KUKA KRL program: MyProgram_176().src

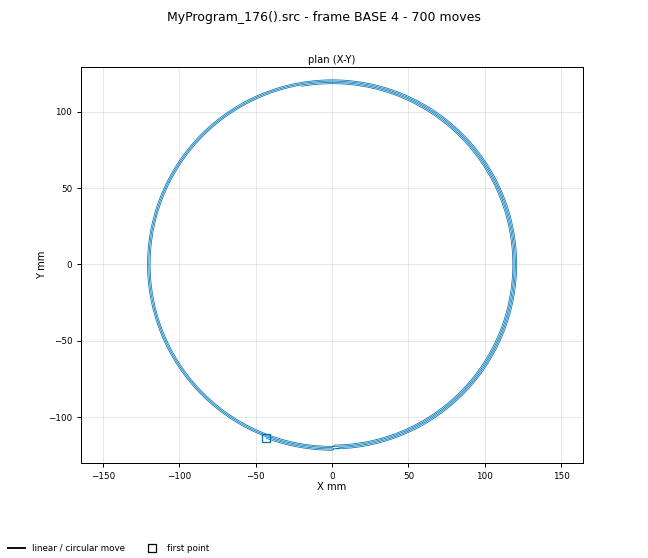
[picture p0: tool path of MyProgram_176().src in frame BASE 4, 700 of 700 moves have a stored position in this frame; points joined in program order, loops and branches not executed]
&ACCESS RVP
&REL 1
&PARAM TEMPLATE = C:\KRC\Roboter\Template\vorgabe
&PARAM EDITMASK = *
DEF MyProgram_176()
; ---- Setting reference (Base) ----
$BASE = BASE_DATA[4]

; --------------------------
; ---- Setting tool (TCP) ----
$TOOL = TOOL_DATA[3]
; --------------------------

$VEL.CP = VEL_APROX_PRINT
Startdeposition()
$VEL.CP = VEL_PRINT
LIN {X -43.076,Y -113.8011,Z 130,A -113.7942,B 24.96,C -1.4605,E1 24.9447,E2 199.9946} C_DIS
LIN {X -39.4863,Y -115.0977,Z 130,A -111.877,B 24.9598,C -1.4645,E1 24.9497,E2 198.0642} C_DIS
LIN {X -36.179,Y -116.1781,Z 130,A -110.3938,B 24.9603,C -1.456,E1 24.9536,E2 196.5985} C_DIS
LIN {X -33.1544,Y -117.077,Z 130,A -108.8854,B 24.9603,C -1.456,E1 24.9577,E2 195.0875} C_DIS
LIN {X -29.6431,Y -118.0168,Z 130,A -107.2113,B 24.9604,C -1.4532,E1 24.9622,E2 193.4176} C_DIS
LIN {X -24.0102,Y -119.2894,Z 130,A -104.7237,B 24.9611,C -1.4411,E1 24.969,E2 190.9557} C_DIS
LIN {X -19.571,Y -120.0977,Z 130,A -102.1105,B 24.9599,C -1.4632,E1 24.9763,E2 188.2874} C_DIS
LIN {X -15.3985,Y -120.7029,Z 130,A -100.2883,B 24.9603,C -1.4551,E1 24.9812,E2 186.483} C_DIS
LIN {X -11.6327,Y -121.1244,Z 130,A -98.1925,B 24.9595,C -1.4697,E1 24.9872,E2 184.3515} C_DIS
LIN {X -8.4115,Y -121.39,Z 130,A -96.7197,B 24.9597,C -1.4674,E1 24.9913,E2 182.8836} C_DIS
LIN {X -3.5905,Y -121.628,Z 130,A -94.6977,B 24.9603,C -1.4557,E1 24.9968,E2 180.8889} C_DIS
LIN {X 0.5177,Y -121.68,Z 130,A -92.4255,B 24.9594,C -1.4722,E1 25.0033,E2 178.5776} C_DIS
LIN {X 0.5177,Y -121.68,Z 130,A -92.4255,B 24.9594,C -1.4722,E1 25.0033,E2 178.5776} C_DIS
Enddeposition()
LIN {X 0.8369,Y -120.8207,Z 130,A -92.2498,B 24.9585,C -1.4882,E1 25.0039,E2 178.364} C_DIS
Startdeposition()
$VEL.CP = VEL_PRINT
LIN {X -2.018,Y -120.82,Z 130,A -95.2101,B 24.9626,C -1.4125,E1 24.9951,E2 181.5038} C_DIS
LIN {X -5.9668,Y -120.6914,Z 130,A -96.5642,B 24.9614,C -1.4362,E1 24.9915,E2 182.8019} C_DIS
LIN {X -11.9573,Y -120.2453,Z 130,A -99.4251,B 24.9614,C -1.4357,E1 24.9835,E2 185.6653} C_DIS
LIN {X -16.915,Y -119.647,Z 130,A -101.5899,B 24.9609,C -1.4455,E1 24.9776,E2 187.8085} C_DIS
LIN {X -21.3625,Y -118.9334,Z 130,A -103.8904,B 24.9612,C -1.4385,E1 24.9712,E2 190.1275} C_DIS
LIN {X -24.4172,Y -118.3441,Z 130,A -105.8718,B 24.9624,C -1.416,E1 24.9656,E2 192.1646} C_DIS
LIN {X -28.0566,Y -117.536,Z 130,A -107.1213,B 24.9611,C -1.4405,E1 24.9624,E2 193.3577} C_DIS
LIN {X -31.1677,Y -116.7485,Z 130,A -108.8063,B 24.9615,C -1.434,E1 24.9578,E2 195.0606} C_DIS
LIN {X -34.3363,Y -115.8557,Z 130,A -110.3107,B 24.9613,C -1.4376,E1 24.9537,E2 196.5589} C_DIS
LIN {X -37.706,Y -114.8044,Z 130,A -111.9297,B 24.9611,C -1.4414,E1 24.9495,E2 198.1718} C_DIS
LIN {X -40.6783,Y -113.7862,Z 130,A -113.4732,B 24.9611,C -1.4402,E1 24.9454,E2 199.721} C_DIS
LIN {X -43.9375,Y -112.5659,Z 130,A -115.4402,B 24.9618,C -1.4276,E1 24.9402,E2 201.7223} C_DIS
LIN {X -49.7061,Y -110.14,Z 130,A -117.7533,B 24.9601,C -1.4602,E1 24.9344,E2 203.9632} C_DIS
LIN {X -52.0013,Y -109.0758,Z 130,A -119.3884,B 24.961,C -1.442,E1 24.9302,E2 205.6457} C_DIS
LIN {X -54.9311,Y -107.6294,Z 130,A -120.8907,B 24.9608,C -1.4461,E1 24.9264,E2 207.1424} C_DIS
LIN {X -58.4415,Y -105.7658,Z 130,A -122.8898,B 24.961,C -1.4435,E1 24.9215,E2 209.1532} C_DIS
LIN {X -61.5431,Y -103.9902,Z 130,A -124.4503,B 24.9605,C -1.452,E1 24.9178,E2 210.6983} C_DIS
LIN {X -64.6206,Y -102.1086,Z 130,A -126.2169,B 24.9605,C -1.452,E1 24.9135,E2 212.4702} C_DIS
LIN {X -67.6234,Y -100.1429,Z 130,A -128.12,B 24.9608,C -1.4459,E1 24.9091,E2 214.3942} C_DIS
LIN {X -73.1245,Y -96.2018,Z 130,A -131.049,B 24.9599,C -1.4639,E1 24.9026,E2 217.2909} C_DIS
LIN {X -75.551,Y -94.3082,Z 130,A -132.6389,B 24.96,C -1.4608,E1 24.899,E2 218.894} C_DIS
LIN {X -78.3065,Y -92.0305,Z 130,A -134.2664,B 24.9597,C -1.4671,E1 24.8956,E2 220.5127} C_DIS
LIN {X -81.1215,Y -89.5618,Z 130,A -136.1792,B 24.9598,C -1.4646,E1 24.8916,E2 222.4392} C_DIS
LIN {X -86.9936,Y -83.8667,Z 130,A -140.8175,B 24.9612,C -1.4401,E1 24.8823,E2 227.1554} C_DIS
LIN {X -90.88,Y -79.639,Z 130,A -142.4074,B 24.9581,C -1.4954,E1 24.8795,E2 228.6207} C_DIS
LIN {X -93.2319,Y -76.8735,Z 130,A -144.4338,B 24.9586,C -1.4861,E1 24.8758,E2 230.6786} C_DIS
LIN {X -97.1767,Y -71.8227,Z 130,A -147.3387,B 24.9579,C -1.4993,E1 24.8709,E2 233.5657} C_DIS
LIN {X -99.5352,Y -68.5169,Z 130,A -149.6462,B 24.9585,C -1.4877,E1 24.8671,E2 235.9122} C_DIS
LIN {X -101.9814,Y -64.8198,Z 130,A -151.6132,B 24.9579,C -1.499,E1 24.8642,E2 237.8621} C_DIS
LIN {X -104.4534,Y -60.7555,Z 130,A -153.9133,B 24.9577,C -1.5032,E1 24.8609,E2 240.1642} C_DIS
LIN {X -106.4444,Y -57.1955,Z 130,A -155.7453,B 24.9571,C -1.5129,E1 24.8584,E2 241.9827} C_DIS
LIN {X -108.1879,Y -53.823,Z 130,A -157.6003,B 24.957,C -1.5157,E1 24.8561,E2 243.8411} C_DIS
LIN {X -109.6658,Y -50.7445,Z 130,A -159.2513,B 24.9568,C -1.5189,E1 24.8541,E2 245.4933} C_DIS
LIN {X -111.2874,Y -47.0815,Z 130,A -161.1444,B 24.9564,C -1.5247,E1 24.852,E2 247.383} C_DIS
LIN {X -112.7082,Y -43.5751,Z 130,A -163.6346,B 24.9578,C -1.5005,E1 24.8494,E2 249.945} C_DIS
LIN {X -114.4356,Y -38.808,Z 130,A -165.0376,B 24.955,C -1.5503,E1 24.8483,E2 251.2373} C_DIS
LIN {X -115.1671,Y -36.5852,Z 130,A -167.6071,B 24.9583,C -1.4919,E1 24.846,E2 253.9606} C_DIS
LIN {X -117.1214,Y -29.7357,Z 130,A -169.9378,B 24.9552,C -1.5464,E1 24.8444,E2 256.1751} C_DIS
LIN {X -118.0083,Y -25.9928,Z 130,A -171.6634,B 24.9546,C -1.5563,E1 24.8433,E2 257.8873} C_DIS
LIN {X -118.6987,Y -22.6313,Z 130,A -173.3036,B 24.9544,C -1.5609,E1 24.8424,E2 259.5262} C_DIS
LIN {X -119.3798,Y -18.7095,Z 130,A -175.2073,B 24.954,C -1.5662,E1 24.8416,E2 261.4286} C_DIS
LIN {X -119.8325,Y -15.5464,Z 130,A -176.7508,B 24.9538,C -1.5698,E1 24.841,E2 262.9726} C_DIS
LIN {X -120.266,Y -11.7482,Z 130,A -178.6463,B 24.9537,C -1.5722,E1 24.8404,E2 264.8739} C_DIS
LIN {X -120.579,Y -7.8922,Z 130,A 179.5994,B 24.9531,C -1.5815,E1 24.8401,E2 266.6164} C_DIS
LIN {X -120.773,Y -3.9289,Z 130,A 177.6956,B 24.9528,C -1.5867,E1 24.8398,E2 268.5194} C_DIS
LIN {X -120.8353,Y -0.6199,Z 130,A 176.1132,B 24.9526,C -1.5913,E1 24.8398,E2 270.1004} C_DIS
LIN {X -120.8018,Y 2.9915,Z 130,A 174.3412,B 24.9524,C -1.5943,E1 24.8398,E2 271.8758} C_DIS
LIN {X -120.6507,Y 6.7033,Z 130,A 172.6318,B 24.9519,C -1.6023,E1 24.8401,E2 273.5764} C_DIS
LIN {X -120.4096,Y 10.165,Z 130,A 171.0115,B 24.9515,C -1.6087,E1 24.8404,E2 275.1911} C_DIS
LIN {X -120.0476,Y 13.7896,Z 130,A 169.1905,B 24.9515,C -1.6104,E1 24.841,E2 277.019} C_DIS
LIN {X -119.5697,Y 17.459,Z 130,A 167.5122,B 24.9509,C -1.6194,E1 24.8416,E2 278.686} C_DIS
LIN {X -119.0095,Y 20.9396,Z 130,A 165.7537,B 24.9508,C -1.6212,E1 24.8424,E2 280.4507} C_DIS
LIN {X -118.3157,Y 24.5557,Z 130,A 164.0299,B 24.9504,C -1.6278,E1 24.8434,E2 282.169} C_DIS
LIN {X -117.5984,Y 27.7942,Z 130,A 161.4095,B 24.9527,C -1.589,E1 24.8452,E2 284.8972} C_DIS
LIN {X -115.9552,Y 34.0007,Z 130,A 159.4245,B 24.9494,C -1.643,E1 24.8466,E2 286.7648} C_DIS
LIN {X -114.9836,Y 37.1522,Z 130,A 157.0631,B 24.9512,C -1.6145,E1 24.8487,E2 289.2078} C_DIS
LIN {X -113.2851,Y 42.0534,Z 130,A 155.3822,B 24.9487,C -1.6549,E1 24.8502,E2 290.8019} C_DIS
LIN {X -111.7939,Y 45.8667,Z 130,A 153.299,B 24.9487,C -1.6549,E1 24.8523,E2 292.8966} C_DIS
LIN {X -108.0583,Y 54.0846,Z 130,A 149.0993,B 24.9477,C -1.6714,E1 24.8573,E2 297.0801} C_DIS
LIN {X -104.2609,Y 61.0851,Z 130,A 145.3907,B 24.9468,C -1.6854,E1 24.8622,E2 300.7749} C_DIS
LIN {X -102.0913,Y 64.6486,Z 130,A 143.1221,B 24.9472,C -1.6787,E1 24.8656,E2 303.0709} C_DIS
LIN {X -98.4997,Y 69.9955,Z 130,A 140.4576,B 24.9456,C -1.7039,E1 24.8697,E2 305.6885} C_DIS
LIN {X -95.4665,Y 74.0798,Z 130,A 137.7866,B 24.9459,C -1.6994,E1 24.8742,E2 308.3832} C_DIS
LIN {X -92.1592,Y 78.1555,Z 130,A 135.5093,B 24.9449,C -1.7151,E1 24.8782,E2 310.6337} C_DIS
LIN {X -88.759,Y 81.9971,Z 130,A 132.9,B 24.9449,C -1.7137,E1 24.883,E2 313.2579} C_DIS
LIN {X -86.6773,Y 84.1949,Z 130,A 131.0333,B 24.9459,C -1.6988,E1 24.8867,E2 315.1682} C_DIS
LIN {X -84.3268,Y 86.55,Z 130,A 129.5286,B 24.9455,C -1.7058,E1 24.8897,E2 316.6627} C_DIS
LIN {X -80.1655,Y 90.4176,Z 130,A 127.1282,B 24.9443,C -1.7247,E1 24.8946,E2 319.0276} C_DIS
LIN {X -77.6232,Y 92.6089,Z 130,A 124.9087,B 24.9458,C -1.7013,E1 24.8995,E2 321.3113} C_DIS
LIN {X -74.2223,Y 95.3568,Z 130,A 123.3101,B 24.9442,C -1.7262,E1 24.9029,E2 322.8566} C_DIS
LIN {X -71.5131,Y 97.4034,Z 130,A 121.4611,B 24.9446,C -1.7193,E1 24.9071,E2 324.7286} C_DIS
LIN {X -67.8075,Y 100.0183,Z 130,A 119.6468,B 24.9434,C -1.7382,E1 24.9112,E2 326.5041} C_DIS
LIN {X -63.7663,Y 102.6424,Z 130,A 116.9018,B 24.9444,C -1.7226,E1 24.9177,E2 329.295} C_DIS
LIN {X -60.5945,Y 104.5468,Z 130,A 115.1497,B 24.9442,C -1.7259,E1 24.922,E2 331.0445} C_DIS
LIN {X -57.4725,Y 106.2942,Z 130,A 113.887,B 24.9428,C -1.7477,E1 24.9249,E2 332.2589} C_DIS
LIN {X -54.5356,Y 107.8315,Z 130,A 112.1726,B 24.943,C -1.7441,E1 24.9292,E2 333.9865} C_DIS
LIN {X -50.8976,Y 109.5945,Z 130,A 110.3644,B 24.9425,C -1.7519,E1 24.9337,E2 335.7808} C_DIS
LIN {X -47.2697,Y 111.2081,Z 130,A 108.4188,B 24.9425,C -1.7519,E1 24.9387,E2 337.7309} C_DIS
LIN {X -44.0241,Y 112.5319,Z 130,A 106.7996,B 24.9422,C -1.7561,E1 24.9429,E2 339.3437} C_DIS
LIN {X -37.4229,Y 114.896,Z 130,A 103.7344,B 24.9412,C -1.7718,E1 24.9509,E2 342.3776} C_DIS
LIN {X -34.8453,Y 115.7047,Z 130,A 102.1371,B 24.942,C -1.7592,E1 24.9553,E2 344.0077} C_DIS
LIN {X -31.5071,Y 116.6568,Z 130,A 100.5707,B 24.9416,C -1.7645,E1 24.9594,E2 345.5639} C_DIS
LIN {X -28.4579,Y 117.4381,Z 130,A 99.0662,B 24.9416,C -1.7654,E1 24.9635,E2 347.0683} C_DIS
LIN {X -24.8301,Y 118.2593,Z 130,A 96.1017,B 24.9449,C -1.7139,E1 24.972,E2 350.1586} C_DIS
LIN {X -17.7522,Y 119.5277,Z 130,A 93.9207,B 24.9412,C -1.7707,E1 24.9776,E2 352.2069} C_DIS
LIN {X -9.9639,Y 120.4257,Z 130,A 90.3564,B 24.9406,C -1.7796,E1 24.9875,E2 355.7521} C_DIS
LIN {X -3.9372,Y 120.7728,Z 130,A 87.429,B 24.9408,C -1.7777,E1 24.9957,E2 358.6849} C_DIS
LIN {X 2.7012,Y 120.8075,Z 130,A 84.3293,B 24.9406,C -1.7805,E1 25.0043,E2 361.778} C_DIS
LIN {X 7.9999,Y 120.5717,Z 130,A 81.8264,B 24.9406,C -1.7811,E1 25.0113,E2 364.2787} C_DIS
LIN {X 14.0154,Y 120.0212,Z 130,A 78.8352,B 24.941,C -1.7749,E1 25.0196,E2 367.2827} C_DIS
LIN {X 17.5208,Y 119.5609,Z 130,A 77.1661,B 24.941,C -1.7748,E1 25.0242,E2 368.9506} C_DIS
LIN {X 20.1208,Y 119.1499,Z 130,A 75.8476,B 24.9412,C -1.7712,E1 25.0279,E2 370.2765} C_DIS
LIN {X 25.1832,Y 118.1848,Z 130,A 73.4943,B 24.941,C -1.7742,E1 25.0343,E2 372.6198} C_DIS
LIN {X 29.3936,Y 117.2093,Z 130,A 71.2197,B 24.9418,C -1.7626,E1 25.0405,E2 374.9185} C_DIS
LIN {X 32.9591,Y 116.255,Z 130,A 69.6385,B 24.9413,C -1.7693,E1 25.0447,E2 376.4813} C_DIS
LIN {X 35.9243,Y 115.3732,Z 130,A 68.1589,B 24.9414,C -1.7676,E1 25.0487,E2 377.9623} C_DIS
LIN {X 38.9416,Y 114.3905,Z 130,A 66.502,B 24.942,C -1.7592,E1 25.0531,E2 379.6358} C_DIS
LIN {X 43.7946,Y 112.622,Z 130,A 64.3605,B 24.9412,C -1.7712,E1 25.0587,E2 381.7444} C_DIS
LIN {X 47.1534,Y 111.2571,Z 130,A 62.5315,B 24.9417,C -1.7643,E1 25.0634,E2 383.5858} C_DIS
LIN {X 49.9349,Y 110.0369,Z 130,A 61.0033,B 24.942,C -1.7585,E1 25.0673,E2 385.1239} C_DIS
LIN {X 55.6396,Y 107.2673,Z 130,A 57.8973,B 24.9426,C -1.7499,E1 25.0751,E2 388.2416} C_DIS
LIN {X 58.9636,Y 105.4742,Z 130,A 56.2743,B 24.9422,C -1.7554,E1 25.0791,E2 389.8472} C_DIS
LIN {X 63.1397,Y 103.0296,Z 130,A 54.0038,B 24.9424,C -1.7531,E1 25.0845,E2 392.1161} C_DIS
LIN {X 65.8525,Y 101.3185,Z 130,A 51.6747,B 24.945,C -1.7125,E1 25.0902,E2 394.5334} C_DIS
LIN {X 70.1284,Y 98.4049,Z 130,A 49.9947,B 24.9429,C -1.7448,E1 25.0938,E2 396.1313} C_DIS
LIN {X 72.8347,Y 96.4195,Z 130,A 48.4007,B 24.9431,C -1.7418,E1 25.0974,E2 397.7266} C_DIS
LIN {X 75.6312,Y 94.2432,Z 130,A 46.6484,B 24.9436,C -1.7352,E1 25.1012,E2 399.488} C_DIS
LIN {X 78.4927,Y 91.8719,Z 130,A 45.0197,B 24.9434,C -1.7382,E1 25.1047,E2 401.1035} C_DIS
LIN {X 83.1482,Y 87.6821,Z 130,A 42.0599,B 24.9437,C -1.7325,E1 25.1108,E2 404.0646} C_DIS
LIN {X 85.565,Y 85.3256,Z 130,A 40.3562,B 24.9443,C -1.7241,E1 25.1142,E2 405.7811} C_DIS
LIN {X 88.5194,Y 82.2578,Z 130,A 38.4664,B 24.9442,C -1.7258,E1 25.1178,E2 407.6586} C_DIS
LIN {X 90.6008,Y 79.9587,Z 130,A 36.8642,B 24.9448,C -1.7161,E1 25.1208,E2 409.2766} C_DIS
LIN {X 93.0238,Y 77.124,Z 130,A 35.1676,B 24.9448,C -1.7154,E1 25.1239,E2 410.9671} C_DIS
LIN {X 95.3788,Y 74.1936,Z 130,A 33.3668,B 24.9452,C -1.7101,E1 25.127,E2 412.7719} C_DIS
LIN {X 97.7429,Y 71.0494,Z 130,A 31.5939,B 24.9452,C -1.7099,E1 25.1299,E2 414.5367} C_DIS
LIN {X 100.4416,Y 67.1823,Z 130,A 29.3918,B 24.9455,C -1.7058,E1 25.1334,E2 416.7378} C_DIS
LIN {X 102.2908,Y 64.3292,Z 130,A 26.8559,B 24.9486,C -1.6569,E1 25.1374,E2 419.3762} C_DIS
LIN {X 105.2879,Y 59.2973,Z 130,A 25.1515,B 24.9458,C -1.7012,E1 25.1396,E2 420.9673} C_DIS
LIN {X 106.4735,Y 57.1418,Z 130,A 23.7123,B 24.9468,C -1.6846,E1 25.1415,E2 422.438} C_DIS
LIN {X 108.2142,Y 53.77,Z 130,A 21.9702,B 24.947,C -1.6824,E1 25.1437,E2 424.1762} C_DIS
LIN {X 109.7481,Y 50.5677,Z 130,A 20.4026,B 24.947,C -1.6832,E1 25.1456,E2 425.7334} C_DIS
LIN {X 111.8091,Y 45.8294,Z 130,A 18.1564,B 24.9467,C -1.686,E1 25.148,E2 427.9606} C_DIS
LIN {X 113.5739,Y 41.2615,Z 130,A 15.7506,B 24.9474,C -1.6749,E1 25.1505,E2 430.3792} C_DIS
LIN {X 114.475,Y 38.691,Z 130,A 14.3368,B 24.9481,C -1.665,E1 25.1517,E2 431.8084} C_DIS
LIN {X 115.4974,Y 35.5239,Z 130,A 12.6878,B 24.9486,C -1.6567,E1 25.1531,E2 433.4677} C_DIS
LIN {X 116.617,Y 31.6547,Z 130,A 10.8737,B 24.9486,C -1.6555,E1 25.1545,E2 435.2742} C_DIS
LIN {X 117.5248,Y 28.1025,Z 130,A 8.6393,B 24.9505,C -1.6257,E1 25.156,E2 437.5659} C_DIS
LIN {X 118.3836,Y 24.225,Z 130,A 7.661,B 24.9481,C -1.6643,E1 25.1565,E2 438.4475} C_DIS
LIN {X 118.8903,Y 21.6022,Z 130,A 5.4208,B 24.9513,C -1.6123,E1 25.1577,E2 440.7971} C_DIS
LIN {X 119.6078,Y 17.1911,Z 130,A 3.0154,B 24.9525,C -1.5916,E1 25.1587,E2 443.2372} C_DIS
LIN {X 120.3033,Y 11.3439,Z 130,A 1.391,B 24.9496,C -1.6399,E1 25.1591,E2 444.7382} C_DIS
LIN {X 120.5914,Y 7.7094,Z 130,A -0.7853,B 24.9513,C -1.6121,E1 25.1596,E2 446.9672} C_DIS
LIN {X 120.8071,Y 2.7026,Z 130,A -3.1872,B 24.9518,C -1.603,E1 25.1598,E2 449.376} C_DIS
LIN {X 120.8349,Y -0.6737,Z 130,A -5.1757,B 24.9533,C -1.5788,E1 25.1598,E2 451.4099} C_DIS
LIN {X 120.7165,Y -5.3935,Z 130,A -6.7524,B 24.9518,C -1.604,E1 25.1596,E2 452.9178} C_DIS
LIN {X 120.432,Y -9.8834,Z 130,A -9.2672,B 24.9533,C -1.5781,E1 25.1591,E2 455.4785} C_DIS
LIN {X 120.0831,Y -13.4863,Z 130,A -10.9402,B 24.9535,C -1.5746,E1 25.1585,E2 457.15} C_DIS
LIN {X 119.6677,Y -16.769,Z 130,A -12.7265,B 24.9545,C -1.5588,E1 25.1578,E2 458.9629} C_DIS
LIN {X 118.9665,Y -21.1784,Z 130,A -14.1691,B 24.9529,C -1.5852,E1 25.1572,E2 460.3351} C_DIS
LIN {X 118.405,Y -24.1205,Z 130,A -15.6612,B 24.9534,C -1.577,E1 25.1564,E2 461.8377} C_DIS
LIN {X 117.649,Y -27.5748,Z 130,A -17.2985,B 24.9536,C -1.5735,E1 25.1554,E2 463.4737} C_DIS
LIN {X 116.5549,Y -31.8843,Z 130,A -19.7071,B 24.9549,C -1.5518,E1 25.1536,E2 465.9195} C_DIS
LIN {X 115.1104,Y -36.7604,Z 130,A -21.8943,B 24.9547,C -1.5552,E1 25.1518,E2 468.0864} C_DIS
LIN {X 112.9222,Y -43.0132,Z 130,A -24.9075,B 24.9549,C -1.5516,E1 25.149,E2 471.0912} C_DIS
LIN {X 111.4747,Y -46.637,Z 130,A -27.5616,B 24.9575,C -1.5063,E1 25.1461,E2 473.8372} C_DIS
LIN {X 109.2269,Y -51.6866,Z 130,A -29.3123,B 24.9555,C -1.541,E1 25.1441,E2 475.4969} C_DIS
LIN {X 107.4928,Y -55.1985,Z 130,A -31.2357,B 24.956,C -1.5321,E1 25.1417,E2 477.431} C_DIS
LIN {X 104.5166,Y -60.647,Z 130,A -34.261,B 24.9568,C -1.5193,E1 25.1376,E2 480.4707} C_DIS
LIN {X 102.1156,Y -64.6097,Z 130,A -36.2375,B 24.9565,C -1.5238,E1 25.1347,E2 482.4266} C_DIS
LIN {X 99.789,Y -68.1462,Z 130,A -38.7448,B 24.9582,C -1.4935,E1 25.1307,E2 484.9928} C_DIS
LIN {X 97.6721,Y -71.1461,Z 130,A -40.9439,B 24.9597,C -1.4665,E1 25.127,E2 487.2452} C_DIS
LIN {X 94.0738,Y -75.8402,Z 130,A -42.8999,B 24.9578,C -1.5001,E1 25.1237,E2 489.1125} C_DIS
LIN {X 89.52,Y -81.1677,Z 130,A -46.9455,B 24.9603,C -1.4563,E1 25.1161,E2 493.2434} C_DIS
LIN {X 85.807,Y -85.0807,Z 130,A -48.6974,B 24.9585,C -1.489,E1 25.1129,E2 494.9105} C_DIS
LIN {X 81.3874,Y -89.3184,Z 130,A -51.464,B 24.9585,C -1.4887,E1 25.1073,E2 497.6666} C_DIS
LIN {X 76.2591,Y -93.7343,Z 130,A -55.6715,B 24.9615,C -1.4331,E1 25.098,E2 501.9891} C_DIS
LIN {X 71.5574,Y -97.3709,Z 130,A -57.9633,B 24.9605,C -1.4523,E1 25.093,E2 504.2273} C_DIS
LIN {X 68.6596,Y -99.436,Z 130,A -59.1332,B 24.9593,C -1.4738,E1 25.0905,E2 505.3424} C_DIS
LIN {X 66.3148,Y -101.0145,Z 130,A -60.9519,B 24.9607,C -1.448,E1 25.0861,E2 507.216} C_DIS
LIN {X 63.3988,Y -102.8704,Z 130,A -62.6823,B 24.9611,C -1.4405,E1 25.0819,E2 508.9587} C_DIS
LIN {X 60.1197,Y -104.8196,Z 130,A -63.6191,B 24.959,C -1.4792,E1 25.0799,E2 509.8012} C_DIS
LIN {X 57.4223,Y -106.3214,Z 130,A -65.3981,B 24.96,C -1.4613,E1 25.0755,E2 511.6174} C_DIS
LIN {X 54.763,Y -107.7154,Z 130,A -66.8713,B 24.9603,C -1.4565,E1 25.0718,E2 513.0978} C_DIS
LIN {X 51.9658,Y -109.0928,Z 130,A -69.5341,B 24.9634,C -1.3978,E1 25.0648,E2 515.8924} C_DIS
LIN {X 45.4408,Y -111.9672,Z 130,A -71.5249,B 24.9601,C -1.4587,E1 25.06,E2 517.7346} C_DIS
LIN {X 39.7455,Y -114.1135,Z 130,A -74.882,B 24.9616,C -1.4323,E1 25.0511,E2 521.1472} C_DIS
LIN {X 35.0777,Y -115.6357,Z 130,A -77.1138,B 24.9615,C -1.434,E1 25.0451,E2 523.3708} C_DIS
LIN {X 31.3737,Y -116.6929,Z 130,A -78.7627,B 24.9611,C -1.4404,E1 25.0407,E2 525.0018} C_DIS
LIN {X 27.4643,Y -117.6746,Z 130,A -80.6829,B 24.9613,C -1.4381,E1 25.0355,E2 526.9247} C_DIS
LIN {X 24.1785,Y -118.3931,Z 130,A -82.9029,B 24.9629,C -1.4073,E1 25.0293,E2 529.2147} C_DIS
LIN {X 19.5282,Y -119.249,Z 130,A -84.3513,B 24.961,C -1.4428,E1 25.0255,E2 530.5778} C_DIS
LIN {X 16.3727,Y -119.7233,Z 130,A -86.3388,B 24.9623,C -1.4194,E1 25.0199,E2 532.6188} C_DIS
LIN {X 13.1382,Y -120.1217,Z 130,A -87.4533,B 24.9612,C -1.4387,E1 25.0169,E2 533.6869} C_DIS
LIN {X 6.275,Y -120.6743,Z 130,A -90.7049,B 24.9612,C -1.4377,E1 25.0079,E2 536.9393} C_DIS
LIN {X 0.8369,Y -120.8207,Z 130,A -92.2444,B 24.9586,C -1.486,E1 25.004,E2 538.3639} C_DIS
Enddeposition()
LIN {X 0.8369,Y -120.8207,Z 130,A -92.2444,B 24.9586,C -1.486,E1 25.004,E2 538.3639} C_DIS
Startdeposition()
$VEL.CP = VEL_PRINT
LIN {X 6.5039,Y -119.8162,Z 130,A -88.9736,B 24.9562,C -1.5281,E1 25.0133,E2 534.9944} C_DIS
LIN {X 12.9507,Y -119.2925,Z 130,A -86.9934,B 24.9591,C -1.4771,E1 25.0184,E2 533.1363} C_DIS
LIN {X 18.4281,Y -118.5691,Z 130,A -84.139,B 24.9585,C -1.4891,E1 25.0264,E2 530.2559} C_DIS
LIN {X 23.9345,Y -117.5814,Z 130,A -81.5882,B 24.9587,C -1.4856,E1 25.0334,E2 527.7164} C_DIS
LIN {X 27.1502,Y -116.8807,Z 130,A -80.0523,B 24.9587,C -1.4854,E1 25.0375,E2 526.183} C_DIS
LIN {X 30.9453,Y -115.9342,Z 130,A -78.1094,B 24.9584,C -1.4909,E1 25.0428,E2 524.23} C_DIS
LIN {X 34.5242,Y -114.9194,Z 130,A -76.3874,B 24.9584,C -1.4904,E1 25.0474,E2 522.5124} C_DIS
LIN {X 37.3657,Y -114.0273,Z 130,A -74.1716,B 24.9561,C -1.5304,E1 25.0536,E2 520.2061} C_DIS
LIN {X 42.4968,Y -112.2151,Z 130,A -72.3887,B 24.9582,C -1.4945,E1 25.058,E2 518.5118} C_DIS
LIN {X 46.0571,Y -110.803,Z 130,A -70.5774,B 24.9581,C -1.4962,E1 25.0627,E2 516.7006} C_DIS
LIN {X 52.0417,Y -108.1198,Z 130,A -67.4338,B 24.9578,C -1.5017,E1 25.0707,E2 513.5519} C_DIS
LIN {X 55.5917,Y -106.3387,Z 130,A -65.5145,B 24.9575,C -1.506,E1 25.0754,E2 511.6276} C_DIS
LIN {X 59.4379,Y -104.2378,Z 130,A -63.6639,B 24.958,C -1.4981,E1 25.0799,E2 509.8013} C_DIS
LIN {X 61.3807,Y -103.1056,Z 130,A -61.6541,B 24.9552,C -1.5457,E1 25.085,E2 507.6851} C_DIS
LIN {X 65.7777,Y -100.3574,Z 130,A -59.8947,B 24.957,C -1.5155,E1 25.0889,E2 506.0029} C_DIS
LIN {X 69.2496,Y -97.9949,Z 130,A -57.7751,B 24.9564,C -1.5252,E1 25.0938,E2 503.8677} C_DIS
LIN {X 74.4542,Y -94.0999,Z 130,A -54.8659,B 24.9566,C -1.5224,E1 25.1003,E2 500.9757} C_DIS
LIN {X 77.3844,Y -91.7071,Z 130,A -53.1711,B 24.9566,C -1.521,E1 25.1039,E2 499.2907} C_DIS
LIN {X 79.9878,Y -89.4437,Z 130,A -51.5346,B 24.9565,C -1.5243,E1 25.1073,E2 497.6528} C_DIS
LIN {X 84.8501,Y -84.8481,Z 130,A -48.2821,B 24.9559,C -1.5348,E1 25.1139,E2 494.3889} C_DIS
LIN {X 89.5758,Y -79.8402,Z 130,A -44.353,B 24.9535,C -1.575,E1 25.1215,E2 490.3824} C_DIS
LIN {X 92.5554,Y -76.3668,Z 130,A -42.709,B 24.9548,C -1.5539,E1 25.1243,E2 488.7957} C_DIS
LIN {X 94.6457,Y -73.7621,Z 130,A -40.691,B 24.9533,C -1.5792,E1 25.1279,E2 486.7274} C_DIS
LIN {X 97.0751,Y -70.5324,Z 130,A -39.0741,B 24.9539,C -1.569,E1 25.1305,E2 485.1424} C_DIS
LIN {X 99.4513,Y -67.1393,Z 130,A -37.2891,B 24.9541,C -1.5651,E1 25.1333,E2 483.3756} C_DIS
LIN {X 101.4734,Y -64.0444,Z 130,A -35.6903,B 24.9543,C -1.5619,E1 25.1356,E2 481.7922} C_DIS
LIN {X 103.6666,Y -60.4316,Z 130,A -32.8628,B 24.9515,C -1.6081,E1 25.1398,E2 478.8703} C_DIS
LIN {X 106.0318,Y -56.1743,Z 130,A -31.2681,B 24.9533,C -1.5786,E1 25.1418,E2 477.3535} C_DIS
LIN {X 107.5334,Y -53.2428,Z 130,A -29.717,B 24.9531,C -1.5823,E1 25.1437,E2 475.8019} C_DIS
LIN {X 109.7932,Y -48.414,Z 130,A -27.2149,B 24.9528,C -1.5879,E1 25.1467,E2 473.3003} C_DIS
LIN {X 111.0584,Y -45.4345,Z 130,A -25.6302,B 24.9524,C -1.5947,E1 25.1484,E2 471.7083} C_DIS
LIN {X 112.2392,Y -42.4332,Z 130,A -24.1036,B 24.9521,C -1.5988,E1 25.1499,E2 470.1803} C_DIS
LIN {X 113.9931,Y -37.4712,Z 130,A -21.5812,B 24.9516,C -1.6072,E1 25.1522,E2 467.6524} C_DIS
LIN {X 114.9984,Y -34.2579,Z 130,A -19.9341,B 24.9512,C -1.6144,E1 25.1536,E2 465.9978} C_DIS
LIN {X 116.1617,Y -30.0784,Z 130,A -17.9335,B 24.951,C -1.6175,E1 25.155,E2 464.0013} C_DIS
LIN {X 116.9905,Y -26.6748,Z 130,A -16.1961,B 24.9505,C -1.6261,E1 25.1561,E2 462.2537} C_DIS
LIN {X 117.8009,Y -22.8292,Z 130,A -14.4442,B 24.9505,C -1.6261,E1 25.1571,E2 460.5123} C_DIS
LIN {X 118.308,Y -20.0372,Z 130,A -12.323,B 24.9478,C -1.6688,E1 25.1581,E2 458.3025} C_DIS
LIN {X 119.0724,Y -14.8432,Z 130,A -10.4886,B 24.9494,C -1.6433,E1 25.1587,E2 456.5393} C_DIS
LIN {X 119.4099,Y -11.8299,Z 130,A -8.5637,B 24.9476,C -1.6719,E1 25.1593,E2 454.5583} C_DIS
LIN {X 119.7636,Y -7.4382,Z 130,A -7.1074,B 24.9492,C -1.6464,E1 25.1596,E2 453.1708} C_DIS
LIN {X 119.9809,Y -1.7386,Z 130,A -4.3448,B 24.9485,C -1.6572,E1 25.1598,E2 450.399} C_DIS
LIN {X 119.9682,Y 2.4259,Z 130,A -1.9376,B 24.9468,C -1.6847,E1 25.1597,E2 447.9415} C_DIS
LIN {X 119.8331,Y 6.1988,Z 130,A -0.1113,B 24.9464,C -1.6917,E1 25.1594,E2 446.1094} C_DIS
LIN {X 119.565,Y 10.1366,Z 130,A 1.4041,B 24.9471,C -1.6794,E1 25.1591,E2 444.6321} C_DIS
LIN {X 119.2131,Y 13.658,Z 130,A 3.4648,B 24.9456,C -1.7034,E1 25.1584,E2 442.527} C_DIS
LIN {X 118.6785,Y 17.72,Z 130,A 5.1451,B 24.9461,C -1.6958,E1 25.1578,E2 440.8744} C_DIS
LIN {X 117.9021,Y 22.3036,Z 130,A 7.2282,B 24.9461,C -1.6961,E1 25.1567,E2 438.8029} C_DIS
LIN {X 117.3081,Y 25.2417,Z 130,A 8.7616,B 24.9455,C -1.7057,E1 25.1558,E2 437.2558} C_DIS
LIN {X 116.2726,Y 29.6471,Z 130,A 10.6727,B 24.9458,C -1.7,E1 25.1546,E2 435.369} C_DIS
LIN {X 115.4843,Y 32.5824,Z 130,A 12.165,B 24.9454,C -1.7066,E1 25.1534,E2 433.8698} C_DIS
LIN {X 114.3401,Y 36.3988,Z 130,A 14.0581,B 24.9451,C -1.7119,E1 25.1519,E2 431.9749} C_DIS
LIN {X 113.3434,Y 39.3907,Z 130,A 15.4299,B 24.9452,C -1.7099,E1 25.1507,E2 430.6157} C_DIS
LIN {X 111.559,Y 44.1918,Z 130,A 17.8886,B 24.9447,C -1.7178,E1 25.1482,E2 428.152} C_DIS
LIN {X 109.6568,Y 48.7236,Z 130,A 20.2927,B 24.9441,C -1.7275,E1 25.1456,E2 425.7383} C_DIS
LIN {X 108.1415,Y 51.9965,Z 130,A 21.9729,B 24.9439,C -1.7304,E1 25.1436,E2 424.0603} C_DIS
LIN {X 106.5374,Y 55.2129,Z 130,A 23.8202,B 24.9432,C -1.7416,E1 25.1412,E2 422.1963} C_DIS
LIN {X 104.4763,Y 59.0192,Z 130,A 26.2798,B 24.9415,C -1.7667,E1 25.1378,E2 419.6903} C_DIS
LIN {X 102.3827,Y 62.5786,Z 130,A 27.6907,B 24.943,C -1.7444,E1 25.1358,E2 418.3391} C_DIS
LIN {X 100.344,Y 65.7981,Z 130,A 29.5092,B 24.9427,C -1.7492,E1 25.1331,E2 416.5186} C_DIS
LIN {X 98.7619,Y 68.1503,Z 130,A 31.0473,B 24.9418,C -1.7617,E1 25.1306,E2 414.9586} C_DIS
LIN {X 96.0615,Y 71.9058,Z 130,A 33.0552,B 24.9421,C -1.7574,E1 25.1273,E2 412.9704} C_DIS
LIN {X 94.0524,Y 74.5143,Z 130,A 34.6417,B 24.9418,C -1.762,E1 25.1246,E2 411.3805} C_DIS
LIN {X 91.4546,Y 77.6808,Z 130,A 36.5575,B 24.9416,C -1.7647,E1 25.1212,E2 409.4672} C_DIS
LIN {X 89.3382,Y 80.1056,Z 130,A 38.1254,B 24.9413,C -1.7698,E1 25.1183,E2 407.8942} C_DIS
LIN {X 87.0907,Y 82.5447,Z 130,A 39.6353,B 24.9413,C -1.7698,E1 25.1154,E2 406.391} C_DIS
LIN {X 84.5295,Y 85.1649,Z 130,A 41.2875,B 24.9413,C -1.7689,E1 25.1122,E2 404.7479} C_DIS
LIN {X 82.0889,Y 87.5194,Z 130,A 43.5789,B 24.9389,C -1.8048,E1 25.1074,E2 402.3811} C_DIS
LIN {X 78.9295,Y 90.3789,Z 130,A 44.9931,B 24.9407,C -1.7789,E1 25.1046,E2 401.0337} C_DIS
LIN {X 76.6174,Y 92.3472,Z 130,A 46.492,B 24.9403,C -1.7841,E1 25.1013,E2 399.5284} C_DIS
LIN {X 73.5252,Y 94.8282,Z 130,A 48.4223,B 24.94,C -1.7894,E1 25.0971,E2 397.5926} C_DIS
LIN {X 70.9387,Y 96.7777,Z 130,A 49.8331,B 24.9402,C -1.7857,E1 25.094,E2 396.1957} C_DIS
LIN {X 66.9086,Y 99.6075,Z 130,A 52.3228,B 24.9395,C -1.7962,E1 25.0882,E2 393.6896} C_DIS
LIN {X 63.8499,Y 101.5948,Z 130,A 54.0245,B 24.9395,C -1.7971,E1 25.0842,E2 391.9913} C_DIS
LIN {X 61.0925,Y 103.2759,Z 130,A 55.7301,B 24.9388,C -1.8072,E1 25.0801,E2 390.2671} C_DIS
LIN {X 57.2326,Y 105.4639,Z 130,A 57.641,B 24.9392,C -1.8004,E1 25.0755,E2 388.378} C_DIS
LIN {X 54.8566,Y 106.7195,Z 130,A 59.2066,B 24.9382,C -1.8154,E1 25.0715,E2 386.781} C_DIS
LIN {X 50.687,Y 108.7614,Z 130,A 61.0821,B 24.9391,C -1.802,E1 25.0669,E2 384.9422} C_DIS
LIN {X 47.7179,Y 110.0967,Z 130,A 62.681,B 24.9389,C -1.8059,E1 25.0628,E2 383.3381} C_DIS
LIN {X 43.1826,Y 111.9554,Z 130,A 65.3462,B 24.9377,C -1.8235,E1 25.0558,E2 380.6371} C_DIS
LIN {X 38.4379,Y 113.6695,Z 130,A 67.3528,B 24.9388,C -1.8068,E1 25.0506,E2 378.6741} C_DIS
LIN {X 35.7611,Y 114.54,Z 130,A 68.7853,B 24.9385,C -1.812,E1 25.0467,E2 377.2319} C_DIS
LIN {X 32.601,Y 115.479,Z 130,A 70.4068,B 24.9382,C -1.8154,E1 25.0424,E2 375.6052} C_DIS
LIN {X 28.7137,Y 116.5067,Z 130,A 72.2699,B 24.9383,C -1.8139,E1 25.0374,E2 373.7483} C_DIS
LIN {X 25.7053,Y 117.207,Z 130,A 73.5633,B 24.9388,C -1.8063,E1 25.0339,E2 372.4748} C_DIS
LIN {X 22.1661,Y 117.9286,Z 130,A 75.4805,B 24.9382,C -1.8159,E1 25.0286,E2 370.5371} C_DIS
LIN {X 18.9583,Y 118.4871,Z 130,A 77.1564,B 24.9378,C -1.8221,E1 25.0239,E2 368.8483} C_DIS
LIN {X 15.2018,Y 119.0259,Z 130,A 78.9912,B 24.9377,C -1.8236,E1 25.0188,E2 367.0116} C_DIS
LIN {X 9.3951,Y 119.6243,Z 130,A 81.5904,B 24.9382,C -1.8152,E1 25.0117,E2 364.4337} C_DIS
LIN {X 5.4968,Y 119.8671,Z 130,A 83.5206,B 24.938,C -1.8182,E1 25.0063,E2 362.4972} C_DIS
LIN {X 1.3481,Y 119.9864,Z 130,A 85.8978,B 24.9368,C -1.836,E1 24.9995,E2 360.078} C_DIS
LIN {X -2.285,Y 119.9708,Z 130,A 87.2212,B 24.9381,C -1.8168,E1 24.996,E2 358.8002} C_DIS
LIN {X -5.8073,Y 119.8536,Z 130,A 89.3751,B 24.9367,C -1.8377,E1 24.9898,E2 356.5962} C_DIS
LIN {X -9.693,Y 119.6005,Z 130,A 90.6791,B 24.9385,C -1.8116,E1 24.9864,E2 355.3536} C_DIS
LIN {X -14.7003,Y 119.0909,Z 130,A 93.2525,B 24.9381,C -1.8179,E1 24.9792,E2 352.7636} C_DIS
LIN {X -18.644,Y 118.5357,Z 130,A 94.9707,B 24.9387,C -1.8084,E1 24.9745,E2 351.0665} C_DIS
LIN {X -24.8872,Y 117.3854,Z 130,A 98.1601,B 24.9384,C -1.8129,E1 24.9657,E2 347.8628} C_DIS
LIN {X -28.086,Y 116.6599,Z 130,A 99.6937,B 24.9386,C -1.81,E1 24.9615,E2 346.3341} C_DIS
LIN {X -31.4345,Y 115.802,Z 130,A 101.3362,B 24.9387,C -1.808,E1 24.9571,E2 344.694} C_DIS
LIN {X -35.3705,Y 114.6611,Z 130,A 103.2095,B 24.9391,C -1.8021,E1 24.9521,E2 342.8315} C_DIS
LIN {X -40.8868,Y 112.812,Z 130,A 106.0852,B 24.9391,C -1.8029,E1 24.9445,E2 339.9483} C_DIS
LIN {X -44.6679,Y 111.3704,Z 130,A 108.0753,B 24.9391,C -1.8029,E1 24.9393,E2 337.9542} C_DIS
LIN {X -47.9272,Y 110.0054,Z 130,A 109.5516,B 24.9399,C -1.791,E1 24.9356,E2 336.5025} C_DIS
LIN {X -50.6478,Y 108.7796,Z 130,A 111.0888,B 24.9397,C -1.7938,E1 24.9317,E2 334.9549} C_DIS
LIN {X -53.0354,Y 107.6361,Z 130,A 112.5162,B 24.9393,C -1.799,E1 24.928,E2 333.5115} C_DIS
LIN {X -56.9184,Y 105.6344,Z 130,A 114.5057,B 24.9399,C -1.7912,E1 24.9232,E2 331.535} C_DIS
LIN {X -64.0115,Y 101.4939,Z 130,A 118.6461,B 24.9397,C -1.7935,E1 24.9132,E2 327.3766} C_DIS
LIN {X -67.9622,Y 98.8927,Z 130,A 120.6001,B 24.9409,C -1.7756,E1 24.9087,E2 325.4585} C_DIS
LIN {X -71.4323,Y 96.4162,Z 130,A 122.6834,B 24.9411,C -1.7735,E1 24.904,E2 323.373} C_DIS
LIN {X -73.2482,Y 95.0417,Z 130,A 124.4956,B 24.9391,C -1.8029,E1 24.8999,E2 321.4842} C_DIS
LIN {X -77.0107,Y 92.0204,Z 130,A 126.2499,B 24.941,C -1.7736,E1 24.8962,E2 319.7929} C_DIS
LIN {X -79.6644,Y 89.7332,Z 130,A 127.6712,B 24.942,C -1.7589,E1 24.8933,E2 318.4011} C_DIS
LIN {X -81.6161,Y 87.9629,Z 130,A 129.1305,B 24.9416,C -1.7646,E1 24.8903,E2 316.9223} C_DIS
LIN {X -85.9107,Y 83.7738,Z 130,A 132.044,B 24.942,C -1.7597,E1 24.8845,E2 314.0082} C_DIS
LIN {X -88.1332,Y 81.4305,Z 130,A 133.443,B 24.9426,C -1.7496,E1 24.8818,E2 312.627} C_DIS
LIN {X -90.8313,Y 78.4115,Z 130,A 135.5383,B 24.9425,C -1.7516,E1 24.878,E2 310.5176} C_DIS
LIN {X -93.8714,Y 74.7433,Z 130,A 137.7851,B 24.943,C -1.7444,E1 24.874,E2 308.2776} C_DIS
LIN {X -97.3442,Y 70.1616,Z 130,A 140.5006,B 24.9435,C -1.7355,E1 24.8695,E2 305.57} C_DIS
LIN {X -100.5758,Y 65.4466,Z 130,A 143.2956,B 24.9439,C -1.7306,E1 24.8651,E2 302.7728} C_DIS
LIN {X -102.7984,Y 61.8947,Z 130,A 145.1947,B 24.9445,C -1.7205,E1 24.8624,E2 300.8881} C_DIS
LIN {X -106.1304,Y 55.987,Z 130,A 148.5188,B 24.9449,C -1.7145,E1 24.8579,E2 297.5608} C_DIS
LIN {X -107.7565,Y 52.7926,Z 130,A 151.1702,B 24.9426,C -1.7498,E1 24.8545,E2 294.811} C_DIS
LIN {X -110.2352,Y 47.4002,Z 130,A 153.2031,B 24.9454,C -1.7065,E1 24.8523,E2 292.87} C_DIS
LIN {X -111.5515,Y 44.2111,Z 130,A 154.7426,B 24.946,C -1.6968,E1 24.8507,E2 291.345} C_DIS
LIN {X -112.8535,Y 40.773,Z 130,A 157.4278,B 24.9438,C -1.7312,E1 24.8481,E2 288.5626} C_DIS
LIN {X -114.6975,Y 35.2531,Z 130,A 159.2765,B 24.947,C -1.6825,E1 24.8466,E2 286.8196} C_DIS
LIN {X -116.9349,Y 26.9157,Z 130,A 163.4903,B 24.9475,C -1.673,E1 24.8436,E2 282.6038} C_DIS
LIN {X -117.7664,Y 23.0085,Z 130,A 165.4034,B 24.9479,C -1.667,E1 24.8425,E2 280.6936} C_DIS
LIN {X -118.3491,Y 19.7915,Z 130,A 167.0018,B 24.9481,C -1.6636,E1 24.8418,E2 279.0941} C_DIS
LIN {X -118.9467,Y 15.813,Z 130,A 168.9092,B 24.9486,C -1.6567,E1 24.841,E2 277.1917} C_DIS
LIN {X -119.3372,Y 12.5235,Z 130,A 170.4594,B 24.949,C -1.6502,E1 24.8406,E2 275.6477} C_DIS
LIN {X -119.6341,Y 9.2724,Z 130,A 172.1268,B 24.949,C -1.6497,E1 24.8402,E2 273.9715} C_DIS
LIN {X -119.8632,Y 5.5868,Z 130,A 173.9118,B 24.9493,C -1.6449,E1 24.8399,E2 272.1872} C_DIS
LIN {X -119.9704,Y 2.3108,Z 130,A 175.4338,B 24.9497,C -1.6379,E1 24.8398,E2 270.6726} C_DIS
LIN {X -119.9858,Y -1.4725,Z 130,A 177.3814,B 24.9497,C -1.6379,E1 24.8398,E2 268.7131} C_DIS
LIN {X -119.8796,Y -5.2064,Z 130,A 179.0507,B 24.9504,C -1.6273,E1 24.84,E2 267.0591} C_DIS
LIN {X -119.649,Y -9.0859,Z 130,A -178.9972,B 24.9504,C -1.6254,E1 24.8404,E2 265.0999} C_DIS
LIN {X -119.3025,Y -12.8558,Z 130,A -177.1768,B 24.9508,C -1.6201,E1 24.8409,E2 263.2812} C_DIS
LIN {X -118.8449,Y -16.5591,Z 130,A -175.4607,B 24.9513,C -1.6116,E1 24.8415,E2 261.5752} C_DIS
LIN {X -118.3264,Y -19.9275,Z 130,A -173.8253,B 24.9516,C -1.6068,E1 24.8422,E2 259.9416} C_DIS
LIN {X -117.6251,Y -23.7219,Z 130,A -171.9958,B 24.952,C -1.6004,E1 24.8432,E2 258.1166} C_DIS
LIN {X -116.9222,Y -26.9708,Z 130,A -170.4696,B 24.9525,C -1.5928,E1 24.8441,E2 256.5995} C_DIS
LIN {X -116.3628,Y -29.2962,Z 130,A -168.065,B 24.9494,C -1.6438,E1 24.846,E2 254.0591} C_DIS
LIN {X -114.4244,Y -36.134,Z 130,A -165.7144,B 24.9527,C -1.588,E1 24.8477,E2 251.8279} C_DIS
LIN {X -111.8828,Y -43.3675,Z 130,A -162.1254,B 24.9536,C -1.5739,E1 24.8511,E2 248.2523} C_DIS
LIN {X -110.6253,Y -46.4787,Z 130,A -160.5707,B 24.954,C -1.5672,E1 24.8528,E2 246.7051} C_DIS
LIN {X -109.2656,Y -49.5918,Z 130,A -158.8898,B 24.9541,C -1.565,E1 24.8547,E2 245.02} C_DIS
LIN {X -107.6421,Y -53.0233,Z 130,A -157.0395,B 24.9543,C -1.5615,E1 24.8569,E2 243.1682} C_DIS
LIN {X -106.0415,Y -56.1559,Z 130,A -155.5139,B 24.955,C -1.5501,E1 24.8589,E2 241.6615} C_DIS
LIN {X -104.1141,Y -59.6531,Z 130,A -153.1173,B 24.954,C -1.5661,E1 24.8622,E2 239.2141} C_DIS
LIN {X -102.451,Y -62.4664,Z 130,A -151.8703,B 24.9551,C -1.5483,E1 24.864,E2 238.0032} C_DIS
LIN {X -100.3797,Y -65.744,Z 130,A -150.2337,B 24.9559,C -1.5341,E1 24.8664,E2 236.3921} C_DIS
LIN {X -98.51,Y -68.5127,Z 130,A -148.4103,B 24.9556,C -1.5399,E1 24.8693,E2 234.5459} C_DIS
LIN {X -96.3497,Y -71.5201,Z 130,A -146.0405,B 24.9543,C -1.5619,E1 24.8733,E2 232.1123} C_DIS
LIN {X -93.5875,Y -75.0995,Z 130,A -144.4492,B 24.956,C -1.5317,E1 24.876,E2 230.5855} C_DIS
LIN {X -91.5028,Y -77.6242,Z 130,A -142.9267,B 24.9564,C -1.5262,E1 24.8787,E2 229.0691} C_DIS
LIN {X -89.693,Y -79.7093,Z 130,A -141.0655,B 24.9552,C -1.5471,E1 24.8823,E2 227.1498} C_DIS
LIN {X -86.892,Y -82.7556,Z 130,A -139.5013,B 24.9565,C -1.5244,E1 24.8852,E2 225.6326} C_DIS
LIN {X -84.9618,Y -84.7351,Z 130,A -137.6738,B 24.9553,C -1.5441,E1 24.8889,E2 223.7507} C_DIS
LIN {X -81.7702,Y -87.8192,Z 130,A -136.0282,B 24.9568,C -1.5186,E1 24.8921,E2 222.1589} C_DIS
LIN {X -79.0843,Y -90.2437,Z 130,A -134.4277,B 24.9573,C -1.5096,E1 24.8954,E2 220.5736} C_DIS
LIN {X -76.6438,Y -92.3253,Z 130,A -132.8254,B 24.9573,C -1.5097,E1 24.8989,E2 218.9647} C_DIS
LIN {X -73.4435,Y -94.8912,Z 130,A -131.1528,B 24.9582,C -1.4934,E1 24.9025,E2 217.3248} C_DIS
LIN {X -70.9822,Y -96.7458,Z 130,A -128.837,B 24.9562,C -1.5285,E1 24.9079,E2 214.9172} C_DIS
LIN {X -67.3912,Y -99.2807,Z 130,A -127.3979,B 24.9581,C -1.4954,E1 24.911,E2 213.552} C_DIS
LIN {X -65.0791,Y -100.8118,Z 130,A -125.9794,B 24.958,C -1.4975,E1 24.9144,E2 212.1239} C_DIS
LIN {X -62.7522,Y -102.2772,Z 130,A -124.6089,B 24.958,C -1.4981,E1 24.9176,E2 210.7478} C_DIS
LIN {X -59.7542,Y -104.056,Z 130,A -123.0152,B 24.9583,C -1.4925,E1 24.9215,E2 209.1626} C_DIS
LIN {X -56.5517,Y -105.8331,Z 130,A -121.1159,B 24.958,C -1.4969,E1 24.9262,E2 207.2475} C_DIS
LIN {X -53.1614,Y -107.5737,Z 130,A -119.406,B 24.9584,C -1.4896,E1 24.9304,E2 205.5503} C_DIS
LIN {X -49.554,Y -109.2826,Z 130,A -117.7521,B 24.9592,C -1.476,E1 24.9345,E2 203.9245} C_DIS
LIN {X -46.0241,Y -110.8169,Z 130,A -115.7359,B 24.9589,C -1.4821,E1 24.9397,E2 201.8893} C_DIS
LIN {X -42.8317,Y -112.0883,Z 130,A -113.9962,B 24.9587,C -1.485,E1 24.9443,E2 200.1389} C_DIS
LIN {X -39.5437,Y -113.2897,Z 130,A -112.3539,B 24.9588,C -1.4822,E1 24.9486,E2 198.5} C_DIS
LIN {X -35.885,Y -114.5016,Z 130,A -110.5251,B 24.959,C -1.4802,E1 24.9534,E2 196.6726} C_DIS
LIN {X -32.7785,Y -115.4287,Z 130,A -108.966,B 24.959,C -1.4796,E1 24.9576,E2 195.1123} C_DIS
LIN {X -29.1564,Y -116.3987,Z 130,A -107.123,B 24.959,C -1.4809,E1 24.9626,E2 193.2635} C_DIS
LIN {X -24.8022,Y -117.4033,Z 130,A -104.9025,B 24.9587,C -1.4839,E1 24.9687,E2 191.0332} C_DIS
LIN {X -21.2184,Y -118.1016,Z 130,A -103.2635,B 24.9591,C -1.4785,E1 24.9732,E2 189.4053} C_DIS
LIN {X -18.4819,Y -118.5608,Z 130,A -101.8589,B 24.9589,C -1.4818,E1 24.9771,E2 187.9916} C_DIS
LIN {X -11.9988,Y -119.3922,Z 130,A -98.8233,B 24.9591,C -1.4773,E1 24.9855,E2 184.9647} C_DIS
LIN {X -6.3429,Y -119.8251,Z 130,A -96.3451,B 24.9597,C -1.4665,E1 24.9923,E2 182.5109} C_DIS
LIN {X -0.2156,Y -119.9935,Z 130,A -93.2838,B 24.9593,C -1.4732,E1 25.0009,E2 179.4336} C_DIS
LIN {X -0.2156,Y -119.9935,Z 130,A -93.2838,B 24.9593,C -1.4732,E1 25.0009,E2 179.4336} C_DIS
Enddeposition()
LIN {X 0.8082,Y -119.1444,Z 130,A -93.2501,B 24.9597,C -1.4669,E1 25.001,E2 179.4147} C_DIS
Startdeposition()
$VEL.CP = VEL_PRINT
LIN {X -3.5599,Y -119.0952,Z 130,A -95.7995,B 24.9608,C -1.446,E1 24.9937,E2 182.0138} C_DIS
LIN {X -7.82,Y -118.8917,Z 130,A -97.5526,B 24.9601,C -1.4594,E1 24.9889,E2 183.7356} C_DIS
LIN {X -10.927,Y -118.6463,Z 130,A -99.1211,B 24.9603,C -1.4564,E1 24.9845,E2 185.3121} C_DIS
LIN {X -14.6865,Y -118.2413,Z 130,A -100.9305,B 24.9603,C -1.457,E1 24.9795,E2 187.1212} C_DIS
LIN {X -18.2664,Y -117.7399,Z 130,A -102.6876,B 24.9603,C -1.4566,E1 24.9746,E2 188.8807} C_DIS
LIN {X -22.2333,Y -117.056,Z 130,A -104.5257,B 24.96,C -1.4617,E1 24.9696,E2 190.7087} C_DIS
LIN {X -25.6925,Y -116.3457,Z 130,A -106.3962,B 24.9604,C -1.4547,E1 24.9644,E2 192.598} C_DIS
LIN {X -29.532,Y -115.4306,Z 130,A -108.2157,B 24.9601,C -1.4593,E1 24.9595,E2 194.4091} C_DIS
LIN {X -32.8257,Y -114.538,Z 130,A -109.9324,B 24.9602,C -1.457,E1 24.9549,E2 196.134} C_DIS
LIN {X -36.2563,Y -113.499,Z 130,A -111.6825,B 24.9602,C -1.457,E1 24.9502,E2 197.887} C_DIS
LIN {X -40.1688,Y -112.1753,Z 130,A -113.6169,B 24.96,C -1.461,E1 24.9451,E2 199.8156} C_DIS
LIN {X -43.265,Y -111.0161,Z 130,A -115.2013,B 24.96,C -1.4628,E1 24.941,E2 201.3992} C_DIS
LIN {X -46.6417,Y -109.6406,Z 130,A -117.0148,B 24.96,C -1.462,E1 24.9363,E2 203.2187} C_DIS
LIN {X -50.1696,Y -108.0711,Z 130,A -118.6557,B 24.9593,C -1.4737,E1 24.9322,E2 204.8359} C_DIS
LIN {X -52.3492,Y -107.0341,Z 130,A -120.043,B 24.9598,C -1.4651,E1 24.9286,E2 206.2472} C_DIS
LIN {X -56.0076,Y -105.1655,Z 130,A -122.0082,B 24.9596,C -1.4681,E1 24.9238,E2 208.2106} C_DIS
LIN {X -59.1625,Y -103.4224,Z 130,A -123.5675,B 24.9591,C -1.4782,E1 24.92,E2 209.7506} C_DIS
LIN {X -61.3895,Y -102.1176,Z 130,A -124.8327,B 24.9591,C -1.4789,E1 24.917,E2 211.0178} C_DIS
LIN {X -64.274,Y -100.3255,Z 130,A -126.5434,B 24.9591,C -1.4781,E1 24.9129,E2 212.7359} C_DIS
LIN {X -67.3841,Y -98.2661,Z 130,A -129.2413,B 24.9611,C -1.4419,E1 24.9065,E2 215.5289} C_DIS
LIN {X -72.0469,Y -94.8997,Z 130,A -131.2043,B 24.9589,C -1.4814,E1 24.9023,E2 217.4051} C_DIS
LIN {X -75.4058,Y -92.2526,Z 130,A -133.3051,B 24.9588,C -1.4833,E1 24.8977,E2 219.5092} C_DIS
LIN {X -78.1766,Y -89.9157,Z 130,A -134.9459,B 24.9583,C -1.4911,E1 24.8943,E2 221.1377} C_DIS
LIN {X -81.2797,Y -87.1217,Z 130,A -137.1466,B 24.9586,C -1.4869,E1 24.8897,E2 223.3574} C_DIS
LIN {X -84.4962,Y -84.0052,Z 130,A -139.1789,B 24.958,C -1.4967,E1 24.8857,E2 225.3748} C_DIS
LIN {X -87.1075,Y -81.2948,Z 130,A -141.138,B 24.9582,C -1.4944,E1 24.8819,E2 227.3481} C_DIS
LIN {X -89.9928,Y -78.0883,Z 130,A -143.0852,B 24.9576,C -1.5046,E1 24.8783,E2 229.2797} C_DIS
LIN {X -92.421,Y -75.1981,Z 130,A -144.5813,B 24.9566,C -1.5225,E1 24.8757,E2 230.7399} C_DIS
LIN {X -95.7789,Y -70.8739,Z 130,A -147.3909,B 24.9566,C -1.5214,E1 24.8709,E2 233.5656} C_DIS
LIN {X -97.322,Y -68.7393,Z 130,A -149.015,B 24.9573,C -1.5094,E1 24.8682,E2 235.2263} C_DIS
LIN {X -100.1094,Y -64.6107,Z 130,A -151.1944,B 24.9564,C -1.5248,E1 24.8649,E2 237.3799} C_DIS
LIN {X -102.0666,Y -61.4734,Z 130,A -153.9346,B 24.9585,C -1.4892,E1 24.8608,E2 240.219} C_DIS
LIN {X -105.0832,Y -56.1613,Z 130,A -155.9989,B 24.9559,C -1.5338,E1 24.8582,E2 242.1879} C_DIS
LIN {X -106.7706,Y -52.8808,Z 130,A -157.7964,B 24.9557,C -1.5378,E1 24.8559,E2 243.9855} C_DIS
LIN {X -108.578,Y -49.063,Z 130,A -159.7457,B 24.9552,C -1.5471,E1 24.8536,E2 245.9233} C_DIS
LIN {X -110.123,Y -45.4934,Z 130,A -161.7213,B 24.9551,C -1.5481,E1 24.8515,E2 247.9075} C_DIS
LIN {X -112.1399,Y -40.266,Z 130,A -164.4091,B 24.9546,C -1.5564,E1 24.8488,E2 250.5906} C_DIS
LIN {X -113.3609,Y -36.6832,Z 130,A -166.1998,B 24.9542,C -1.5632,E1 24.8473,E2 252.3754} C_DIS
LIN {X -114.4249,Y -33.223,Z 130,A -167.863,B 24.9537,C -1.5718,E1 24.8459,E2 254.0278} C_DIS
LIN {X -115.6031,Y -28.856,Z 130,A -170.2369,B 24.9538,C -1.5702,E1 24.8442,E2 256.4192} C_DIS
LIN {X -116.4662,Y -25.1402,Z 130,A -172.0638,B 24.9534,C -1.5763,E1 24.8431,E2 258.2423} C_DIS
LIN {X -117.233,Y -21.2793,Z 130,A -173.7387,B 24.9525,C -1.5914,E1 24.8423,E2 259.8911} C_DIS
LIN {X -117.6422,Y -18.8984,Z 130,A -175.2118,B 24.9531,C -1.5821,E1 24.8416,E2 261.3952} C_DIS
LIN {X -118.1976,Y -15.0249,Z 130,A -177.0234,B 24.9526,C -1.5911,E1 24.8409,E2 263.1962} C_DIS
LIN {X -118.6135,Y -11.2825,Z 130,A -178.7667,B 24.952,C -1.5997,E1 24.8404,E2 264.9293} C_DIS
LIN {X -118.8524,Y -8.4017,Z 130,A 179.814,B 24.9519,C -1.603,E1 24.8401,E2 266.3493} C_DIS
LIN {X -119.0469,Y -4.9205,Z 130,A 178.1259,B 24.9516,C -1.608,E1 24.8399,E2 268.0357} C_DIS
LIN {X -119.1439,Y -1.109,Z 130,A 176.3359,B 24.9511,C -1.6158,E1 24.8398,E2 269.8179} C_DIS
LIN {X -119.1373,Y 1.6995,Z 130,A 175.0927,B 24.9505,C -1.6246,E1 24.8398,E2 271.0475} C_DIS
LIN {X -119.0668,Y 4.4588,Z 130,A 173.5023,B 24.9509,C -1.618,E1 24.84,E2 272.6632} C_DIS
LIN {X -118.8752,Y 8.0638,Z 130,A 171.837,B 24.9504,C -1.6267,E1 24.8402,E2 274.318} C_DIS
LIN {X -118.5326,Y 12.1022,Z 130,A 169.8836,B 24.95,C -1.6329,E1 24.8407,E2 276.2683} C_DIS
LIN {X -118.1409,Y 15.4625,Z 130,A 168.2971,B 24.9496,C -1.6398,E1 24.8413,E2 277.8476} C_DIS
LIN {X -117.6152,Y 19.062,Z 130,A 166.4192,B 24.9496,C -1.6402,E1 24.8421,E2 279.7358} C_DIS
LIN {X -117.0129,Y 22.4572,Z 130,A 164.8568,B 24.949,C -1.6496,E1 24.8429,E2 281.2852} C_DIS
LIN {X -116.2042,Y 26.3283,Z 130,A 162.3781,B 24.9501,C -1.6319,E1 24.8444,E2 283.8206} C_DIS
LIN {X -115.209,Y 30.3929,Z 130,A 160.7724,B 24.9487,C -1.6551,E1 24.8455,E2 285.3804} C_DIS
LIN {X -114.2449,Y 33.8298,Z 130,A 159.1698,B 24.948,C -1.6653,E1 24.8467,E2 286.9678} C_DIS
LIN {X -113.3413,Y 36.7436,Z 130,A 157.3627,B 24.9486,C -1.6559,E1 24.8483,E2 288.8078} C_DIS
LIN {X -111.5694,Y 41.8184,Z 130,A 155.0633,B 24.9474,C -1.6758,E1 24.8504,E2 291.0727} C_DIS
LIN {X -110.3657,Y 44.8973,Z 130,A 153.5167,B 24.9469,C -1.6826,E1 24.852,E2 292.6118} C_DIS
LIN {X -108.1385,Y 50.0248,Z 130,A 150.7657,B 24.9466,C -1.6882,E1 24.8551,E2 295.3645} C_DIS
LIN {X -106.648,Y 53.1281,Z 130,A 149.1125,B 24.9463,C -1.6933,E1 24.8571,E2 297.0145} C_DIS
LIN {X -104.9996,Y 56.3182,Z 130,A 147.2437,B 24.9463,C -1.6925,E1 24.8596,E2 298.8951} C_DIS
LIN {X -102.3772,Y 60.954,Z 130,A 144.7055,B 24.9458,C -1.701,E1 24.8631,E2 301.4264} C_DIS
LIN {X -100.3549,Y 64.2282,Z 130,A 143.201,B 24.9445,C -1.7208,E1 24.8653,E2 302.8913} C_DIS
LIN {X -98.3686,Y 67.2327,Z 130,A 141.0919,B 24.9452,C -1.7099,E1 24.8686,E2 305.037} C_DIS
LIN {X -96.0655,Y 70.4825,Z 130,A 139.1683,B 24.9449,C -1.7149,E1 24.8718,E2 306.9581} C_DIS
LIN {X -93.588,Y 73.7405,Z 130,A 137.5696,B 24.9435,C -1.7357,E1 24.8744,E2 308.5147} C_DIS
LIN {X -89.6489,Y 78.482,Z 130,A 134.708,B 24.9427,C -1.7478,E1 24.8795,E2 311.3606} C_DIS
LIN {X -87.7369,Y 80.6138,Z 130,A 132.8929,B 24.9437,C -1.7328,E1 24.883,E2 313.2196} C_DIS
LIN {X -85.2824,Y 83.2092,Z 130,A 130.3494,B 24.9457,C -1.7025,E1 24.8881,E2 315.8461} C_DIS
LIN {X -81.4033,Y 87.0054,Z 130,A 128.447,B 24.9434,C -1.7383,E1 24.8918,E2 317.671} C_DIS
LIN {X -78.4062,Y 89.7151,Z 130,A 126.5784,B 24.9429,C -1.746,E1 24.8957,E2 319.5288} C_DIS
LIN {X -76.1966,Y 91.5993,Z 130,A 124.7951,B 24.9437,C -1.7328,E1 24.8996,E2 321.3504} C_DIS
LIN {X -73.3156,Y 93.9238,Z 130,A 123.3146,B 24.9427,C -1.7493,E1 24.9027,E2 322.7972} C_DIS
LIN {X -70.5437,Y 96.0207,Z 130,A 121.5252,B 24.9427,C -1.7478,E1 24.9068,E2 324.5964} C_DIS
LIN {X -67.2203,Y 98.3769,Z 130,A 119.7237,B 24.942,C -1.7585,E1 24.9109,E2 326.3786} C_DIS
LIN {X -64.9631,Y 99.8832,Z 130,A 118.5155,B 24.9416,C -1.7651,E1 24.9137,E2 327.575} C_DIS
LIN {X -60.5563,Y 102.6123,Z 130,A 115.3485,B 24.9432,C -1.7411,E1 24.9214,E2 330.8089} C_DIS
LIN {X -56.6571,Y 104.8157,Z 130,A 114.239,B 24.94,C -1.7896,E1 24.9238,E2 331.8063} C_DIS
LIN {X -53.7481,Y 106.338,Z 130,A 112.2237,B 24.9411,C -1.7733,E1 24.9289,E2 333.8658} C_DIS
LIN {X -50.3503,Y 107.987,Z 130,A 110.3801,B 24.9409,C -1.775,E1 24.9336,E2 335.71} C_DIS
LIN {X -46.8007,Y 109.5736,Z 130,A 108.6296,B 24.9404,C -1.783,E1 24.938,E2 337.4459} C_DIS
LIN {X -43.7871,Y 110.8111,Z 130,A 106.8289,B 24.9409,C -1.775,E1 24.9427,E2 339.2694} C_DIS
LIN {X -39.976,Y 112.2433,Z 130,A 105.0549,B 24.9402,C -1.7856,E1 24.9473,E2 341.0219} C_DIS
LIN {X -36.0833,Y 113.555,Z 130,A 102.9837,B 24.9404,C -1.7838,E1 24.9528,E2 343.1013} C_DIS
LIN {X -33.0504,Y 114.4743,Z 130,A 101.3447,B 24.9406,C -1.7805,E1 24.9573,E2 344.7508} C_DIS
LIN {X -29.5953,Y 115.4143,Z 130,A 99.8545,B 24.9398,C -1.7924,E1 24.9612,E2 346.215} C_DIS
LIN {X -25.6019,Y 116.3655,Z 130,A 97.9969,B 24.9393,C -1.7993,E1 24.9662,E2 348.0586} C_DIS
LIN {X -22.1006,Y 117.0816,Z 130,A 95.9774,B 24.9401,C -1.7875,E1 24.9718,E2 350.1083} C_DIS
LIN {X -18.8431,Y 117.6507,Z 130,A 94.3687,B 24.9401,C -1.7878,E1 24.9763,E2 351.7178} C_DIS
LIN {X -15.6721,Y 118.1138,Z 130,A 92.9053,B 24.9398,C -1.7923,E1 24.9803,E2 353.1718} C_DIS
LIN {X -11.9766,Y 118.5457,Z 130,A 91.028,B 24.94,C -1.7893,E1 24.9855,E2 355.0573} C_DIS
LIN {X -7.7553,Y 118.8961,Z 130,A 89.0924,B 24.9396,C -1.7947,E1 24.9909,E2 356.9809} C_DIS
LIN {X -3.6592,Y 119.0922,Z 130,A 87.1174,B 24.9396,C -1.7953,E1 24.9964,E2 358.955} C_DIS
LIN {X -0.03,Y 119.1502,Z 130,A 85.1157,B 24.9403,C -1.7842,E1 25.0021,E2 360.9829} C_DIS
LIN {X 4.8063,Y 119.0518,Z 130,A 83.169,B 24.9392,C -1.8014,E1 25.0074,E2 362.8884} C_DIS
LIN {X 7.8028,Y 118.8929,Z 130,A 81.818,B 24.9389,C -1.8056,E1 25.0111,E2 364.2291} C_DIS
LIN {X 9.8411,Y 118.7418,Z 130,A 80.6372,B 24.9395,C -1.7966,E1 25.0145,E2 365.4305} C_DIS
LIN {X 13.5588,Y 118.3748,Z 130,A 78.825,B 24.9395,C -1.7956,E1 25.0195,E2 367.2438} C_DIS
LIN {X 16.7941,Y 117.9589,Z 130,A 77.1604,B 24.9399,C -1.7909,E1 25.0241,E2 368.9182} C_DIS
LIN {X 20.3947,Y 117.3921,Z 130,A 75.55,B 24.9395,C -1.7967,E1 25.0285,E2 370.5132} C_DIS
LIN {X 22.88,Y 116.9315,Z 130,A 74.1989,B 24.9399,C -1.7901,E1 25.0323,E2 371.8784} C_DIS
LIN {X 26.6629,Y 116.1269,Z 130,A 72.4204,B 24.9398,C -1.7928,E1 25.0371,E2 373.648} C_DIS
LIN {X 29.7319,Y 115.3792,Z 130,A 70.9516,B 24.9397,C -1.7942,E1 25.041,E2 375.1114} C_DIS
LIN {X 33.1858,Y 114.4359,Z 130,A 69.2179,B 24.9397,C -1.7924,E1 25.0457,E2 376.8465} C_DIS
LIN {X 36.5571,Y 113.4017,Z 130,A 67.4857,B 24.94,C -1.7895,E1 25.0503,E2 378.5825} C_DIS
LIN {X 39.2241,Y 112.5072,Z 130,A 66.0579,B 24.9403,C -1.7848,E1 25.0541,E2 380.0185} C_DIS
LIN {X 43.2146,Y 111.0359,Z 130,A 63.9825,B 24.9405,C -1.7815,E1 25.0596,E2 382.0974} C_DIS
LIN {X 47.2304,Y 109.3883,Z 130,A 62.1695,B 24.9398,C -1.7918,E1 25.0642,E2 383.8816} C_DIS
LIN {X 49.6954,Y 108.2919,Z 130,A 60.8068,B 24.9401,C -1.7873,E1 25.0676,E2 385.2518} C_DIS
LIN {X 52.6887,Y 106.8658,Z 130,A 59.1029,B 24.9406,C -1.7803,E1 25.072,E2 386.9678} C_DIS
LIN {X 55.9333,Y 105.2047,Z 130,A 57.3516,B 24.9408,C -1.778,E1 25.0763,E2 388.7195} C_DIS
LIN {X 59.3925,Y 103.2903,Z 130,A 55.4732,B 24.9408,C -1.7763,E1 25.0809,E2 390.5962} C_DIS
LIN {X 62.8218,Y 101.2417,Z 130,A 53.7829,B 24.9403,C -1.7841,E1 25.0849,E2 392.2628} C_DIS
LIN {X 65.5553,Y 99.493,Z 130,A 51.9629,B 24.9413,C -1.7695,E1 25.0892,E2 394.1115} C_DIS
LIN {X 68.1705,Y 97.7198,Z 130,A 50.3988,B 24.9416,C -1.7649,E1 25.0928,E2 395.6812} C_DIS
LIN {X 71.4544,Y 95.3448,Z 130,A 48.5923,B 24.9414,C -1.7681,E1 25.0968,E2 397.4738} C_DIS
LIN {X 73.967,Y 93.409,Z 130,A 47.0281,B 24.9417,C -1.7634,E1 25.1003,E2 399.0431} C_DIS
LIN {X 77.0882,Y 90.8504,Z 130,A 45.0871,B 24.942,C -1.7596,E1 25.1045,E2 400.9856} C_DIS
LIN {X 82.9692,Y 85.5138,Z 130,A 41.3527,B 24.9422,C -1.7557,E1 25.1121,E2 404.7141} C_DIS
LIN {X 85.9562,Y 82.5102,Z 130,A 39.2286,B 24.9428,C -1.7471,E1 25.1163,E2 406.8494} C_DIS
LIN {X 88.5953,Y 79.6699,Z 130,A 37.4104,B 24.9429,C -1.7451,E1 25.1197,E2 408.6645} C_DIS
LIN {X 90.7501,Y 77.2061,Z 130,A 35.8723,B 24.9431,C -1.7431,E1 25.1225,E2 410.2003} C_DIS
LIN {X 93.047,Y 74.4251,Z 130,A 34.0159,B 24.9437,C -1.7331,E1 25.1258,E2 412.0717} C_DIS
LIN {X 95.2717,Y 71.5517,Z 130,A 32.437,B 24.9435,C -1.7368,E1 25.1285,E2 413.6343} C_DIS
LIN {X 97.4925,Y 68.4975,Z 130,A 30.4555,B 24.9443,C -1.7243,E1 25.1317,E2 415.6357} C_DIS
LIN {X 99.5438,Y 65.4782,Z 130,A 28.8196,B 24.9443,C -1.7254,E1 25.1342,E2 417.2608} C_DIS
LIN {X 101.7804,Y 61.9442,Z 130,A 26.8579,B 24.9444,C -1.7224,E1 25.1371,E2 419.2196} C_DIS
LIN {X 103.7627,Y 58.5657,Z 130,A 24.9609,B 24.9448,C -1.7166,E1 25.1398,E2 421.1206} C_DIS
LIN {X 105.362,Y 55.6346,Z 130,A 23.3794,B 24.945,C -1.7133,E1 25.1419,E2 422.7015} C_DIS
LIN {X 106.8356,Y 52.7497,Z 130,A 21.8108,B 24.9453,C -1.7084,E1 25.1438,E2 424.2734} C_DIS
LIN {X 108.5104,Y 49.213,Z 130,A 19.9469,B 24.9456,C -1.7038,E1 25.146,E2 426.138} C_DIS
LIN {X 109.9019,Y 46.0216,Z 130,A 18.3041,B 24.9458,C -1.7004,E1 25.1478,E2 427.7798} C_DIS
LIN {X 111.2261,Y 42.7248,Z 130,A 16.7143,B 24.9458,C -1.7011,E1 25.1495,E2 429.3592} C_DIS
LIN {X 112.2304,Y 40.013,Z 130,A 15.1205,B 24.9467,C -1.6871,E1 25.151,E2 430.9771} C_DIS
LIN {X 113.3966,Y 36.5728,Z 130,A 13.4598,B 24.9467,C -1.6859,E1 25.1524,E2 432.6311} C_DIS
LIN {X 114.4543,Y 33.1208,Z 130,A 11.6511,B 24.9473,C -1.6771,E1 25.1539,E2 434.4504} C_DIS
LIN {X 115.3944,Y 29.6729,Z 130,A 10.0954,B 24.9471,C -1.6796,E1 25.155,E2 435.9911} C_DIS
LIN {X 116.399,Y 25.4484,Z 130,A 8.0381,B 24.9475,C -1.6746,E1 25.1563,E2 438.0483} C_DIS
LIN {X 116.9097,Y 22.9935,Z 130,A 6.8455,B 24.9477,C -1.6714,E1 25.157,E2 439.2415} C_DIS
LIN {X 117.5138,Y 19.6687,Z 130,A 5.213,B 24.948,C -1.6659,E1 25.1578,E2 440.8776} C_DIS
LIN {X 118.0836,Y 15.905,Z 130,A 3.2692,B 24.9487,C -1.6544,E1 25.1585,E2 442.8368} C_DIS
LIN {X 118.5039,Y 12.3764,Z 130,A 1.7509,B 24.9485,C -1.6582,E1 25.159,E2 444.3372} C_DIS
LIN {X 118.7936,Y 9.1929,Z 130,A 0.1058,B 24.9491,C -1.648,E1 25.1594,E2 445.9966} C_DIS
LIN {X 119.0619,Y 4.5728,Z 130,A -2.2012,B 24.9498,C -1.6367,E1 25.1597,E2 448.3165} C_DIS
LIN {X 119.146,Y 0.7673,Z 130,A -3.8885,B 24.9498,C -1.6377,E1 25.1597,E2 449.9914} C_DIS
LIN {X 119.1132,Y -2.9638,Z 130,A -5.9073,B 24.9508,C -1.6209,E1 25.1597,E2 452.0378} C_DIS
LIN {X 118.9032,Y -7.6504,Z 130,A -8.1371,B 24.9511,C -1.6148,E1 25.1593,E2 454.2688} C_DIS
LIN {X 118.4894,Y -12.5146,Z 130,A -10.2596,B 24.9509,C -1.6181,E1 25.1588,E2 456.371} C_DIS
LIN {X 118.0455,Y -16.1844,Z 130,A -12.2242,B 24.9518,C -1.6031,E1 25.1581,E2 458.3592} C_DIS
LIN {X 117.322,Y -20.7844,Z 130,A -14.2713,B 24.9518,C -1.6052,E1 25.1571,E2 460.3895} C_DIS
LIN {X 116.6969,Y -24.0456,Z 130,A -15.8538,B 24.952,C -1.6007,E1 25.1563,E2 461.9733} C_DIS
LIN {X 115.8237,Y -27.9519,Z 130,A -17.7661,B 24.9523,C -1.595,E1 25.1551,E2 463.8878} C_DIS
LIN {X 114.9842,Y -31.2249,Z 130,A -19.309,B 24.9524,C -1.5938,E1 25.154,E2 465.4247} C_DIS
LIN {X 114.019,Y -34.5911,Z 130,A -21.1572,B 24.9532,C -1.5804,E1 25.1525,E2 467.2941} C_DIS
LIN {X 112.7479,Y -38.5291,Z 130,A -23.024,B 24.9532,C -1.5801,E1 25.1509,E2 469.1511} C_DIS
LIN {X 111.6981,Y -41.4769,Z 130,A -24.6553,B 24.9539,C -1.5691,E1 25.1493,E2 470.7989} C_DIS
LIN {X 110.491,Y -44.5894,Z 130,A -26.148,B 24.9539,C -1.5696,E1 25.1478,E2 472.2822} C_DIS
LIN {X 108.9509,Y -48.2337,Z 130,A -28.1194,B 24.9544,C -1.5604,E1 25.1456,E2 474.2647} C_DIS
LIN {X 107.1467,Y -52.1176,Z 130,A -30.1546,B 24.9547,C -1.5553,E1 25.1431,E2 476.3009} C_DIS
LIN {X 105.5086,Y -55.3563,Z 130,A -31.9803,B 24.9552,C -1.5461,E1 25.1408,E2 478.1385} C_DIS
LIN {X 103.549,Y -58.9422,Z 130,A -33.7921,B 24.9552,C -1.5477,E1 25.1383,E2 479.9372} C_DIS
LIN {X 101.5678,Y -62.2942,Z 130,A -35.6836,B 24.9555,C -1.5413,E1 25.1356,E2 481.8342} C_DIS
LIN {X 99.7833,Y -65.1149,Z 130,A -37.109,B 24.9553,C -1.5454,E1 25.1335,E2 483.2428} C_DIS
LIN {X 98.3478,Y -67.2634,Z 130,A -38.5258,B 24.9559,C -1.5334,E1 25.1312,E2 484.6808} C_DIS
LIN {X 96.4782,Y -69.9188,Z 130,A -40.1977,B 24.9565,C -1.5237,E1 25.1285,E2 486.3674} C_DIS
LIN {X 93.5542,Y -73.7832,Z 130,A -42.2943,B 24.9562,C -1.5287,E1 25.1249,E2 488.4424} C_DIS
LIN {X 91.2934,Y -76.5646,Z 130,A -44.2102,B 24.957,C -1.5148,E1 25.1215,E2 490.3823} C_DIS
LIN {X 87.2451,Y -81.1484,Z 130,A -46.9979,B 24.957,C -1.5145,E1 25.1163,E2 493.1582} C_DIS
LIN {X 84.7979,Y -83.6998,Z 130,A -48.587,B 24.957,C -1.5156,E1 25.1132,E2 494.7378} C_DIS
LIN {X 81.284,Y -87.1175,Z 130,A -51.1913,B 24.958,C -1.498,E1 25.1079,E2 497.3728} C_DIS
LIN {X 77.7203,Y -90.3119,Z 130,A -53.354,B 24.9579,C -1.4993,E1 25.1034,E2 499.524} C_DIS
LIN {X 74.7223,Y -92.8066,Z 130,A -55.2079,B 24.9581,C -1.4961,E1 25.0994,E2 501.3784} C_DIS
LIN {X 72.5056,Y -94.5481,Z 130,A -56.532,B 24.9581,C -1.4947,E1 25.0964,E2 502.7011} C_DIS
LIN {X 69.6311,Y -96.6857,Z 130,A -58.284,B 24.9584,C -1.4896,E1 25.0925,E2 504.4589} C_DIS
LIN {X 66.2919,Y -99.0056,Z 130,A -60.0804,B 24.9582,C -1.4932,E1 25.0884,E2 506.2407} C_DIS
LIN {X 61.6771,Y -101.9428,Z 130,A -62.8378,B 24.9589,C -1.4821,E1 25.0818,E2 509.0156} C_DIS
LIN {X 59.2714,Y -103.3598,Z 130,A -64.3047,B 24.9593,C -1.4737,E1 25.0782,E2 510.4978} C_DIS
LIN {X 55.4571,Y -105.4554,Z 130,A -66.1811,B 24.9589,C -1.4803,E1 25.0737,E2 512.3533} C_DIS
LIN {X 52.1176,Y -107.1467,Z 130,A -68.2076,B 24.9597,C -1.4666,E1 25.0685,E2 514.4067} C_DIS
LIN {X 47.6612,Y -109.2005,Z 130,A -70.3198,B 24.9593,C -1.4746,E1 25.0632,E2 516.4948} C_DIS
LIN {X 44.2282,Y -110.6378,Z 130,A -72.2218,B 24.9597,C -1.4667,E1 25.0582,E2 518.4112} C_DIS
LIN {X 40.3256,Y -112.1181,Z 130,A -74.3404,B 24.9601,C -1.4588,E1 25.0527,E2 520.544} C_DIS
LIN {X 35.7408,Y -113.6625,Z 130,A -76.4681,B 24.9598,C -1.4652,E1 25.0471,E2 522.6525} C_DIS
LIN {X 32.5006,Y -114.6301,Z 130,A -78.0458,B 24.9598,C -1.4656,E1 25.0428,E2 524.2265} C_DIS
LIN {X 28.785,Y -115.6204,Z 130,A -79.7679,B 24.9595,C -1.4696,E1 25.0382,E2 525.9365} C_DIS
LIN {X 25.6811,Y -116.3482,Z 130,A -81.2597,B 24.9595,C -1.47,E1 25.0342,E2 527.4252} C_DIS
LIN {X 23.6677,Y -116.7744,Z 130,A -82.3779,B 24.9599,C -1.4632,E1 25.0311,E2 528.5583} C_DIS
LIN {X 18.0342,Y -117.7758,Z 130,A -85.1669,B 24.9601,C -1.4593,E1 25.0234,E2 531.3536} C_DIS
LIN {X 14.2039,Y -118.2992,Z 130,A -86.8696,B 24.9598,C -1.4653,E1 25.0187,E2 533.0407} C_DIS
LIN {X 12.1826,Y -118.5242,Z 130,A -88.3205,B 24.961,C -1.4429,E1 25.0145,E2 534.5435} C_DIS
LIN {X 8.8812,Y -118.8185,Z 130,A -89.6953,B 24.9605,C -1.4522,E1 25.0108,E2 535.8957} C_DIS
LIN {X 3.1874,Y -119.1067,Z 130,A -92.3222,B 24.9603,C -1.4564,E1 25.0035,E2 538.5118} C_DIS
LIN {X 0.8082,Y -119.1444,Z 130,A -93.2484,B 24.9597,C -1.4662,E1 25.0009,E2 539.4148} C_DIS
Enddeposition()
LIN {X 0.8082,Y -119.1444,Z 130,A -93.2484,B 24.9597,C -1.4662,E1 25.0009,E2 539.4148} C_DIS
Startdeposition()
$VEL.CP = VEL_PRINT
LIN {X 1.4434,Y -118.2976,Z 130,A -92.5041,B 24.9578,C -1.501,E1 25.0033,E2 538.588} C_DIS
LIN {X 3.9892,Y -118.2375,Z 130,A -91.2409,B 24.9577,C -1.5028,E1 25.0068,E2 537.3208} C_DIS
LIN {X 6.8055,Y -118.1087,Z 130,A -89.8945,B 24.9577,C -1.5025,E1 25.0105,E2 535.9756} C_DIS
LIN {X 9.7874,Y -117.8992,Z 130,A -88.4612,B 24.9577,C -1.5025,E1 25.0145,E2 534.5429} C_DIS
LIN {X 13.0384,Y -117.5858,Z 130,A -86.8803,B 24.9577,C -1.5033,E1 25.0189,E2 532.9611} C_DIS
LIN {X 15.5658,Y -117.2763,Z 130,A -85.6195,B 24.9575,C -1.5055,E1 25.0224,E2 531.6963} C_DIS
LIN {X 18.4224,Y -116.8616,Z 130,A -84.254,B 24.9575,C -1.505,E1 25.0262,E2 530.3334} C_DIS
LIN {X 21.2641,Y -116.378,Z 130,A -82.8274,B 24.9575,C -1.5075,E1 25.0301,E2 528.9023} C_DIS
LIN {X 24.501,Y -115.7416,Z 130,A -81.2649,B 24.9575,C -1.5072,E1 25.0344,E2 527.3423} C_DIS
LIN {X 27.3273,Y -115.107,Z 130,A -79.8655,B 24.9574,C -1.5084,E1 25.0382,E2 525.942} C_DIS
LIN {X 29.8046,Y -114.4889,Z 130,A -78.601,B 24.9572,C -1.5111,E1 25.0416,E2 524.6732} C_DIS
LIN {X 32.492,Y -113.7551,Z 130,A -77.2723,B 24.9572,C -1.5116,E1 25.0452,E2 523.3455} C_DIS
LIN {X 35.7264,Y -112.7832,Z 130,A -75.6529,B 24.9572,C -1.5127,E1 25.0495,E2 521.7263} C_DIS
LIN {X 38.1526,Y -111.984,Z 130,A -74.4167,B 24.957,C -1.5143,E1 25.0528,E2 520.4888} C_DIS
LIN {X 41.2301,Y -110.8895,Z 130,A -72.8464,B 24.957,C -1.5158,E1 25.0569,E2 518.9181} C_DIS
LIN {X 43.9291,Y -109.8483,Z 130,A -71.4452,B 24.9568,C -1.5178,E1 25.0606,E2 517.5153} C_DIS
LIN {X 46.6017,Y -108.7414,Z 130,A -70.0484,B 24.9568,C -1.5197,E1 25.0642,E2 516.1173} C_DIS
LIN {X 48.9335,Y -107.7104,Z 130,A -68.8066,B 24.9566,C -1.522,E1 25.0673,E2 514.8733} C_DIS
LIN {X 51.8587,Y -106.3346,Z 130,A -67.2591,B 24.9566,C -1.5236,E1 25.0712,E2 513.3259} C_DIS
LIN {X 54.0563,Y -105.2325,Z 130,A -66.0192,B 24.9563,C -1.528,E1 25.0743,E2 512.079} C_DIS
LIN {X 56.7405,Y -103.8102,Z 130,A -64.5709,B 24.9562,C -1.5295,E1 25.0779,E2 510.6314} C_DIS
LIN {X 59.5734,Y -102.2127,Z 130,A -63.0372,B 24.9562,C -1.5304,E1 25.0816,E2 509.1002} C_DIS
LIN {X 62.0445,Y -100.7316,Z 130,A -61.6495,B 24.956,C -1.5327,E1 25.0849,E2 507.7114} C_DIS
LIN {X 64.1894,Y -99.3767,Z 130,A -60.4186,B 24.9558,C -1.5352,E1 25.0878,E2 506.4785} C_DIS
LIN {X 66.9253,Y -97.5573,Z 130,A -58.8389,B 24.9557,C -1.5379,E1 25.0915,E2 504.8978} C_DIS
LIN {X 70.1851,Y -95.2369,Z 130,A -56.9063,B 24.9555,C -1.5417,E1 25.0959,E2 502.963} C_DIS
LIN {X 72.219,Y -93.7033,Z 130,A -55.6826,B 24.9553,C -1.5439,E1 25.0986,E2 501.7385} C_DIS
LIN {X 74.5957,Y -91.8226,Z 130,A -54.1645,B 24.955,C -1.5496,E1 25.1019,E2 500.2127} C_DIS
LIN {X 77.0554,Y -89.7694,Z 130,A -52.657,B 24.955,C -1.551,E1 25.1051,E2 498.7077} C_DIS
LIN {X 79.8395,Y -87.3017,Z 130,A -50.8424,B 24.9546,C -1.5559,E1 25.1089,E2 496.8888} C_DIS
LIN {X 82.2302,Y -85.0537,Z 130,A -49.2378,B 24.9544,C -1.5605,E1 25.1121,E2 495.28} C_DIS
LIN {X 85.0544,Y -82.2294,Z 130,A -47.338,B 24.9542,C -1.5636,E1 25.1158,E2 493.3809} C_DIS
LIN {X 87.2691,Y -79.8751,Z 130,A -45.7707,B 24.954,C -1.5677,E1 25.1188,E2 491.8108} C_DIS
LIN {X 89.4384,Y -77.4398,Z 130,A -44.2347,B 24.9538,C -1.5697,E1 25.1217,E2 490.277} C_DIS
LIN {X 91.8012,Y -74.6222,Z 130,A -42.4394,B 24.9535,C -1.5752,E1 25.1249,E2 488.4771} C_DIS
LIN {X 93.7042,Y -72.2179,Z 130,A -40.9613,B 24.9533,C -1.5789,E1 25.1274,E2 486.9972} C_DIS
LIN {X 95.8668,Y -69.3249,Z 130,A -39.2672,B 24.9532,C -1.581,E1 25.1302,E2 485.3063} C_DIS
LIN {X 97.3615,Y -67.207,Z 130,A -38.0167,B 24.953,C -1.5844,E1 25.1322,E2 484.054} C_DIS
LIN {X 99.12,Y -64.5873,Z 130,A -36.4953,B 24.9527,C -1.5884,E1 25.1345,E2 482.5307} C_DIS
LIN {X 100.7168,Y -62.0688,Z 130,A -35.063,B 24.9525,C -1.592,E1 25.1367,E2 481.0972} C_DIS
LIN {X 102.2131,Y -59.5727,Z 130,A -33.6613,B 24.9523,C -1.5957,E1 25.1387,E2 479.6939} C_DIS
LIN {X 103.4693,Y -57.3596,Z 130,A -32.4348,B 24.9521,C -1.5991,E1 25.1403,E2 478.4657} C_DIS
LIN {X 104.837,Y -54.8198,Z 130,A -31.0807,B 24.952,C -1.6012,E1 25.1421,E2 477.1138} C_DIS
LIN {X 106.1689,Y -52.1939,Z 130,A -29.6297,B 24.9516,C -1.6068,E1 25.1439,E2 475.6575} C_DIS
LIN {X 107.4235,Y -49.5606,Z 130,A -28.1969,B 24.9513,C -1.6121,E1 25.1456,E2 474.22} C_DIS
LIN {X 108.6036,Y -46.9181,Z 130,A -26.8363,B 24.9512,C -1.6144,E1 25.1471,E2 472.8612} C_DIS
LIN {X 109.6725,Y -44.3609,Z 130,A -25.487,B 24.9509,C -1.6189,E1 25.1486,E2 471.5087} C_DIS
LIN {X 110.89,Y -41.2287,Z 130,A -23.8869,B 24.9507,C -1.6226,E1 25.1502,E2 469.9087} C_DIS
LIN {X 111.8654,Y -38.5037,Z 130,A -22.4933,B 24.9504,C -1.6267,E1 25.1515,E2 468.5135} C_DIS
LIN {X 112.6679,Y -36.0828,Z 130,A -21.2811,B 24.9502,C -1.6295,E1 25.1525,E2 467.3014} C_DIS
LIN {X 113.6243,Y -32.9535,Z 130,A -19.6925,B 24.9499,C -1.6348,E1 25.1538,E2 465.7096} C_DIS
LIN {X 114.3128,Y -30.4734,Z 130,A -18.4244,B 24.9496,C -1.6399,E1 25.1547,E2 464.4367} C_DIS
LIN {X 115.106,Y -27.3316,Z 130,A -16.8962,B 24.9494,C -1.6429,E1 25.1557,E2 462.9102} C_DIS
LIN {X 115.7409,Y -24.5044,Z 130,A -15.5024,B 24.9492,C -1.647,E1 25.1565,E2 461.5149} C_DIS
LIN {X 116.2419,Y -21.9968,Z 130,A -14.2436,B 24.9489,C -1.652,E1 25.1572,E2 460.2515} C_DIS
LIN {X 116.8023,Y -18.8051,Z 130,A -12.7136,B 24.9487,C -1.6552,E1 25.1579,E2 458.723} C_DIS
LIN {X 117.1834,Y -16.2512,Z 130,A -11.4432,B 24.9483,C -1.6603,E1 25.1584,E2 457.4481} C_DIS
LIN {X 117.5456,Y -13.3817,Z 130,A -10.0813,B 24.9482,C -1.663,E1 25.1589,E2 456.0879} C_DIS
LIN {X 117.869,Y -10.1631,Z 130,A -8.5251,B 24.9479,C -1.6676,E1 25.1593,E2 454.5301} C_DIS
LIN {X 118.1448,Y -6.1521,Z 130,A -6.592,B 24.9475,C -1.6733,E1 25.1596,E2 452.5949} C_DIS
LIN {X 118.2543,Y -3.4419,Z 130,A -5.2225,B 24.9471,C -1.6804,E1 25.1597,E2 451.217} C_DIS
LIN {X 118.3065,Y -0.0025,Z 130,A -3.634,B 24.947,C -1.682,E1 25.1597,E2 449.6341} C_DIS
LIN {X 118.2374,Y 3.9926,Z 130,A -1.6811,B 24.9465,C -1.6892,E1 25.1597,E2 447.6759} C_DIS
LIN {X 118.0856,Y 7.2221,Z 130,A -0.1602,B 24.9463,C -1.6921,E1 25.1594,E2 446.1572} C_DIS
LIN {X 117.8973,Y 9.8111,Z 130,A 1.0925,B 24.9461,C -1.696,E1 25.1591,E2 444.9028} C_DIS
LIN {X 117.5865,Y 13.0311,Z 130,A 2.6489,B 24.9458,C -1.7005,E1 25.1587,E2 443.3449} C_DIS
LIN {X 117.2768,Y 15.5617,Z 130,A 3.9048,B 24.9455,C -1.7055,E1 25.1583,E2 442.0845} C_DIS
LIN {X 116.8616,Y 18.422,Z 130,A 5.2696,B 24.9453,C -1.7083,E1 25.1577,E2 440.7211} C_DIS
LIN {X 116.3683,Y 21.3182,Z 130,A 6.7067,B 24.945,C -1.7135,E1 25.157,E2 439.2802} C_DIS
LIN {X 115.7427,Y 24.4958,Z 130,A 8.2357,B 24.9448,C -1.7166,E1 25.1561,E2 437.753} C_DIS
LIN {X 115.1085,Y 27.3209,Z 130,A 9.6245,B 24.9445,C -1.7203,E1 25.1552,E2 436.3634} C_DIS
LIN {X 114.0203,Y 31.556,Z 130,A 11.7324,B 24.9441,C -1.7264,E1 25.1537,E2 434.2532} C_DIS
LIN {X 113.3109,Y 34.01,Z 130,A 12.991,B 24.9438,C -1.7313,E1 25.1527,E2 432.9904} C_DIS
LIN {X 112.3384,Y 37.1012,Z 130,A 14.5205,B 24.9436,C -1.7341,E1 25.1514,E2 431.4629} C_DIS
LIN {X 111.5038,Y 39.5341,Z 130,A 15.794,B 24.9433,C -1.7392,E1 25.1503,E2 430.1844} C_DIS
LIN {X 110.4973,Y 42.2657,Z 130,A 17.1881,B 24.9431,C -1.7427,E1 25.1489,E2 428.7899} C_DIS
LIN {X 109.3028,Y 45.2693,Z 130,A 18.7161,B 24.9429,C -1.7455,E1 25.1473,E2 427.2639} C_DIS
LIN {X 108.2538,Y 47.7204,Z 130,A 19.9914,B 24.9427,C -1.7485,E1 25.1459,E2 425.9884} C_DIS
LIN {X 106.9498,Y 50.5782,Z 130,A 21.5114,B 24.9424,C -1.7528,E1 25.1441,E2 424.4665} C_DIS
LIN {X 105.679,Y 53.1823,Z 130,A 22.9031,B 24.9422,C -1.7562,E1 25.1423,E2 423.0741} C_DIS
LIN {X 103.8088,Y 56.7431,Z 130,A 24.871,B 24.9418,C -1.7626,E1 25.1397,E2 421.1014} C_DIS
LIN {X 102.2049,Y 59.5865,Z 130,A 26.4071,B 24.9416,C -1.7648,E1 25.1376,E2 419.5682} C_DIS
LIN {X 100.7166,Y 62.0691,Z 130,A 27.8048,B 24.9414,C -1.7683,E1 25.1356,E2 418.1692} C_DIS
LIN {X 99.353,Y 64.2263,Z 130,A 29.0099,B 24.9413,C -1.7701,E1 25.1338,E2 416.9659} C_DIS
LIN {X 97.5596,Y 66.9219,Z 130,A 30.5969,B 24.9409,C -1.7751,E1 25.1313,E2 415.3751} C_DIS
LIN {X 95.8932,Y 69.2884,Z 130,A 32.157,B 24.9402,C -1.7863,E1 25.1287,E2 413.7962} C_DIS
LIN {X 93.7034,Y 72.2189,Z 130,A 33.7527,B 24.9405,C -1.7823,E1 25.1261,E2 412.2176} C_DIS
LIN {X 91.7976,Y 74.6265,Z 130,A 35.2821,B 24.9401,C -1.7879,E1 25.1234,E2 410.682} C_DIS
LIN {X 89.6945,Y 77.1434,Z 130,A 36.8212,B 24.94,C -1.7893,E1 25.1206,E2 409.1466} C_DIS
LIN {X 87.2875,Y 79.8549,Z 130,A 38.6018,B 24.9396,C -1.7945,E1 25.1173,E2 407.3617} C_DIS
LIN {X 85.0669,Y 82.2164,Z 130,A 40.1761,B 24.9394,C -1.7982,E1 25.1142,E2 405.7854} C_DIS
LIN {X 82.749,Y 84.5506,Z 130,A 41.7168,B 24.9394,C -1.7991,E1 25.1112,E2 404.2491} C_DIS
LIN {X 80.1375,Y 87.0282,Z 130,A 43.4848,B 24.939,C -1.8039,E1 25.1076,E2 402.4769} C_DIS
LIN {X 77.8717,Y 89.0612,Z 130,A 44.8979,B 24.939,C -1.804,E1 25.1046,E2 401.0692} C_DIS
LIN {X 75.6125,Y 90.987,Z 130,A 46.344,B 24.9388,C -1.8072,E1 25.1015,E2 399.6211} C_DIS
LIN {X 73.2262,Y 92.9185,Z 130,A 47.8759,B 24.9384,C -1.8121,E1 25.0982,E2 398.0834} C_DIS
LIN {X 70.6068,Y 94.9257,Z 130,A 49.3929,B 24.9385,C -1.8112,E1 25.0948,E2 396.5741} C_DIS
LIN {X 68.3855,Y 96.5374,Z 130,A 50.7414,B 24.9383,C -1.8144,E1 25.0917,E2 395.2227} C_DIS
LIN {X 66.0039,Y 98.1811,Z 130,A 52.1674,B 24.9381,C -1.8179,E1 25.0884,E2 393.7932} C_DIS
LIN {X 63.2936,Y 99.9517,Z 130,A 53.7008,B 24.938,C -1.8188,E1 25.0849,E2 392.2628} C_DIS
LIN {X 59.5834,Y 102.2067,Z 130,A 55.7952,B 24.9378,C -1.8216,E1 25.0798,E2 390.1682} C_DIS
LIN {X 57.3651,Y 103.4663,Z 130,A 56.9935,B 24.9378,C -1.8216,E1 25.0769,E2 388.9733} C_DIS
LIN {X 55.0466,Y 104.7176,Z 130,A 58.3466,B 24.9374,C -1.827,E1 25.0736,E2 387.6115} C_DIS
LIN {X 52.4401,Y 106.0469,Z 130,A 59.7565,B 24.9374,C -1.8285,E1 25.07,E2 386.2018} C_DIS
LIN {X 49.5753,Y 107.4166,Z 130,A 61.2762,B 24.9373,C -1.8295,E1 25.0662,E2 384.6836} C_DIS
LIN {X 46.9297,Y 108.5985,Z 130,A 62.6476,B 24.9373,C -1.8295,E1 25.0627,E2 383.3154} C_DIS
LIN {X 44.2561,Y 109.7152,Z 130,A 64.049,B 24.9372,C -1.831,E1 25.0591,E2 381.9139} C_DIS
LIN {X 41.2283,Y 110.8902,Z 130,A 65.6167,B 24.9371,C -1.8322,E1 25.055,E2 380.3465} C_DIS
LIN {X 38.5081,Y 111.8638,Z 130,A 67.0085,B 24.9371,C -1.8331,E1 25.0513,E2 378.9554} C_DIS
LIN {X 34.6674,Y 113.1115,Z 130,A 68.9949,B 24.9368,C -1.8361,E1 25.046,E2 376.9656} C_DIS
LIN {X 31.8868,Y 113.9266,Z 130,A 70.3676,B 24.9368,C -1.8357,E1 25.0424,E2 375.5961} C_DIS
LIN {X 28.7937,Y 114.7488,Z 130,A 71.9035,B 24.9368,C -1.836,E1 25.0382,E2 374.0619} C_DIS
LIN {X 24.5055,Y 115.7406,Z 130,A 74.0448,B 24.9368,C -1.8376,E1 25.0324,E2 371.9197} C_DIS
LIN {X 21.988,Y 116.2436,Z 130,A 75.3156,B 24.9366,C -1.8394,E1 25.0289,E2 370.6462} C_DIS
LIN {X 18.798,Y 116.8035,Z 130,A 76.8547,B 24.9366,C -1.8386,E1 25.0247,E2 369.1106} C_DIS
LIN {X 16.2732,Y 117.1803,Z 130,A 78.1199,B 24.9366,C -1.8403,E1 25.0211,E2 367.8426} C_DIS
LIN {X 13.401,Y 117.5433,Z 130,A 79.4916,B 24.9366,C -1.8392,E1 25.0174,E2 366.4745} C_DIS
LIN {X 10.1806,Y 117.8674,Z 130,A 81.0595,B 24.9366,C -1.8393,E1 25.013,E2 364.9072} C_DIS
LIN {X 7.2604,Y 118.0834,Z 130,A 82.4758,B 24.9366,C -1.8393,E1 25.0091,E2 363.4916} C_DIS
LIN {X 2.9255,Y 118.2702,Z 130,A 84.5791,B 24.9366,C -1.8392,E1 25.0032,E2 361.3891} C_DIS
LIN {X 0.3775,Y 118.3041,Z 130,A 85.8447,B 24.9366,C -1.8404,E1 24.9996,E2 360.1206} C_DIS
LIN {X -2.56,Y 118.2772,Z 130,A 87.2367,B 24.9366,C -1.8387,E1 24.9958,E2 358.7327} C_DIS
LIN {X -5.7946,Y 118.1644,Z 130,A 88.806,B 24.9366,C -1.8382,E1 24.9914,E2 357.1641} C_DIS
LIN {X -8.3405,Y 118.0104,Z 130,A 90.0417,B 24.9366,C -1.8378,E1 24.9879,E2 355.929} C_DIS
LIN {X -11.2464,Y 117.7691,Z 130,A 91.4849,B 24.9366,C -1.8385,E1 24.9839,E2 354.4836} C_DIS
LIN {X -14.1242,Y 117.4587,Z 130,A 92.8612,B 24.9368,C -1.8365,E1 24.9801,E2 353.1109} C_DIS
LIN {X -16.855,Y 117.0976,Z 130,A 94.2171,B 24.9368,C -1.8367,E1 24.9764,E2 351.7537} C_DIS
LIN {X -19.8729,Y 116.6237,Z 130,A 95.6767,B 24.9369,C -1.8347,E1 24.9724,E2 350.2973} C_DIS
Enddeposition()
END
